LIN {X 0,Y 322.641,Z 978.52,A -85,B 0,C 180,E1 11313.588,E2 11313.588} C_VEL
LIN {X 0,Y 314.07,Z 998.583,A -85,B 0,C 180,E1 11311.867,E2 11311.867} C_VEL
LIN {X 0,Y 304.732,Z 1017.6,A -85,B 0,C 180,E1 11309.836,E2 11309.836} C_VEL
LIN {X 0,Y 294.954,Z 1035.741,A -85,B 0,C 180,E1 11307.468,E2 11307.468} C_VEL
LIN {X 0,Y 285.433,Z 1051.736,A -85,B 0,C 180,E1 11304.898,E2 11304.898} C_VEL
LIN {X 0,Y 275.123,Z 1067.9,A -85,B 0,C 180,E1 11301.721,E2 11301.721} C_VEL
LIN {X 0,Y 265.925,Z 1081.436,A -85,B 0,C 180,E1 11298.438,E2 11298.438} C_VEL
LIN {X 0,Y 256.201,Z 1095.185,A -85,B 0,C 180,E1 11294.314,E2 11294.314} C_VEL
LIN {X 0,Y 248.125,Z 1106.369,A -85,B 0,C 180,E1 11290.148,E2 11290.148} C_VEL
LIN {X 0,Y 240.588,Z 1116.784,A -85,B 0,C 180,E1 11285.288,E2 11285.288} C_VEL
LIN {X 0,Y 234.378,Z 1125.809,A -85,B 0,C 180,E1 11280.002,E2 11280.002} C_VEL
LIN {X 0,Y 229.706,Z 1133.063,A -85,B 0,C 180,E1 11274.427,E2 11274.427} C_VEL
LIN {X 0,Y 226.641,Z 1138.738,A -85,B 0,C 180,E1 11268.788,E2 11268.788} C_VEL
LIN {X 0,Y 224.919,Z 1142.727,A -85,B 0,C 180,E1 11263.105,E2 11263.105} C_VEL
LIN {X 0,Y 224.189,Z 1145.377,A -85,B 0,C 180,E1 11257.432,E2 11257.432} C_VEL
LIN {X 0,Y 224.031,Z 1146.421,A -85,B 0,C 180,E1 11252.303,E2 11252.303} C_VEL
LIN {X 0,Y 224.031,Z 1146.452,A -85,B 0,C 180,E1 11247.954,E2 11247.954} C_VEL
LIN {X 0,Y 224.161,Z 1145.534,A -85,B 0,C 180,E1 11243.083,E2 11243.083} C_VEL
LIN {X 0,Y 224.802,Z 1143.101,A -85,B 0,C 180,E1 11237.413,E2 11237.413} C_VEL
LIN {X 0,Y 226.193,Z 1139.618,A -85,B 0,C 180,E1 11232.242,E2 11232.242} C_VEL
LIN {X 0,Y 229.316,Z 1133.777,A -85,B 0,C 180,E1 11226.078,E2 11226.078} C_VEL
LIN {X 0,Y 233.531,Z 1127.081,A -85,B 0,C 180,E1 11220.785,E2 11220.785} C_VEL
LIN {X 0,Y 239.772,Z 1117.979,A -85,B 0,C 180,E1 11215.236,E2 11215.236} C_VEL
LIN {X 0,Y 247.238,Z 1107.713,A -85,B 0,C 180,E1 11210.285,E2 11210.285} C_VEL
LIN {X 0,Y 255.624,Z 1096.058,A -85,B 0,C 180,E1 11205.875,E2 11205.875} C_VEL
LIN {X 0,Y 265.28,Z 1082.497,A -85,B 0,C 180,E1 11201.731,E2 11201.731} C_VEL
LIN {X 0,Y 274.982,Z 1068.229,A -85,B 0,C 180,E1 11198.243,E2 11198.243} C_VEL
LIN {X 0,Y 285.562,Z 1051.675,A -85,B 0,C 180,E1 11194.983,E2 11194.983} C_VEL
LIN {X 0,Y 294.996,Z 1035.841,A -85,B 0,C 180,E1 11192.44,E2 11192.44} C_VEL
LIN {X 0,Y 304.922,Z 1017.448,A -85,B 0,C 180,E1 11190.041,E2 11190.041} C_VEL
LIN {X 0,Y 313.925,Z 999.165,A -85,B 0,C 180,E1 11188.085,E2 11188.085} C_VEL
LIN {X 0,Y 322.495,Z 979.181,A -85,B 0,C 180,E1 11186.362,E2 11186.362} C_VEL
LIN {X 0,Y 330.224,Z 958.766,A -85,B 0,C 180,E1 11184.929,E2 11184.929} C_VEL
LIN {X 0,Y 336.593,Z 938.741,A -85,B 0,C 180,E1 11183.805,E2 11183.805} C_VEL
LIN {X 0,Y 338.848,Z 930.878,A -85,B 0,C 180,E1 11183.416,E2 11183.416} C_VEL
LIN {X 0,Y 340.313,Z 923.759,A -85,B 0,C 180,E1 11182.949,E2 11182.949} C_VEL
LIN {X 0,Y 342.235,Z 906.193,A -85,B 0,C 180,E1 11181.337,E2 11181.337} C_VEL
LIN {X 0,Y 343.315,Z 898.896,A -85,B 0,C 180,E1 11180.949,E2 11180.949} C_VEL
LIN {X 0,Y 347.119,Z 876.033,A -85,B 0,C 180,E1 11180.35,E2 11180.35} C_VEL
LIN {X 0,Y 351.591,Z 829.528,A -85,B 0,C 180,E1 11179.437,E2 11179.437} C_VEL
LIN {X 0,Y 362.38,Z 710.369,A -85,B 0,C 180,E1 11177.172,E2 11177.172} C_VEL
LIN {X 0,Y 358.599,Z 703.638,A -85,B 0,C 180,E1 11174.534,E2 11174.534} C_VEL
LIN {X 0,Y 355.948,Z 699.091,A -85,B 0,C 180,E1 11172.327,E2 11172.327} C_VEL
LIN {X 0,Y 354.328,Z 696.281,A -85,B 0,C 180,E1 11170.734,E2 11170.734} C_VEL
LIN {X 0,Y 352.108,Z 692.354,A -85,B 0,C 180,E1 11167.999,E2 11167.999} C_VEL
LIN {X 0,Y 350.023,Z 688.483,A -85,B 0,C 180,E1 11163.767,E2 11163.767} C_VEL
LIN {X 0,Y 349.776,Z 687.555,A -85,B 0,C 180,E1 11162.622,E2 11162.622} C_VEL
LIN {X 0,Y 349.89,Z 687.727,A -85,B 0,C 180,E1 11157.38,E2 11157.38} C_VEL
LIN {X 0,Y 351.646,Z 691.826,A -85,B 0,C 180,E1 11153.142,E2 11153.142} C_VEL
LIN {X 0,Y 352.509,Z 693.002,A -85,B 0,C 180,E1 11151.929,E2 11151.929} C_VEL
LIN {X 0,Y 355.354,Z 697.958,A -85,B 0,C 180,E1 11148.723,E2 11148.723} C_VEL
LIN {X 0,Y 357.98,Z 702.565,A -85,B 0,C 180,E1 11146.431,E2 11146.431} C_VEL
LIN {X 0,Y 361.715,Z 709.096,A -85,B 0,C 180,E1 11143.748,E2 11143.748} C_VEL
LIN {X 0,Y 362.516,Z 710.882,A -85,B 0,C 180,E1 11143.207,E2 11143.207} C_VEL
LIN {X 0,Y 346.978,Z 881.346,A -85,B 0,C 180,E1 11139.937,E2 11139.937} C_VEL
LIN {X 0,Y 343.192,Z 905.388,A -85,B 0,C 180,E1 11139.359,E2 11139.359} C_VEL
LIN {X 0,Y 338.384,Z 927.394,A -85,B 0,C 180,E1 11138.689,E2 11138.689} C_VEL
LIN {X 0,Y 332.183,Z 949.393,A -85,B 0,C 180,E1 11137.784,E2 11137.784} C_VEL
LIN {X 0,Y 325.051,Z 970.759,A -85,B 0,C 180,E1 11136.663,E2 11136.663} C_VEL
LIN {X 0,Y 316.962,Z 991.126,A -85,B 0,C 180,E1 11135.298,E2 11135.298} C_VEL
LIN {X 0,Y 307.991,Z 1011.145,A -85,B 0,C 180,E1 11133.638,E2 11133.638} C_VEL
LIN {X 0,Y 298.944,Z 1028.985,A -85,B 0,C 180,E1 11131.801,E2 11131.801} C_VEL
LIN {X 0,Y 288.556,Z 1047.701,A -85,B 0,C 180,E1 11129.436,E2 11129.436} C_VEL
LIN {X 0,Y 278.69,Z 1063.904,A -85,B 0,C 180,E1 11126.901,E2 11126.901} C_VEL
LIN {X 0,Y 267.235,Z 1081.449,A -85,B 0,C 180,E1 11123.495,E2 11123.495} C_VEL
LIN {X 0,Y 257.236,Z 1095.991,A -85,B 0,C 180,E1 11119.971,E2 11119.971} C_VEL
LIN {X 0,Y 247.673,Z 1109.311,A -85,B 0,C 180,E1 11115.938,E2 11115.938} C_VEL
LIN {X 0,Y 238.923,Z 1121.487,A -85,B 0,C 180,E1 11111.392,E2 11111.392} C_VEL
LIN {X 0,Y 231.282,Z 1132.166,A -85,B 0,C 180,E1 11106.318,E2 11106.318} C_VEL
LIN {X 0,Y 225.037,Z 1141.571,A -85,B 0,C 180,E1 11100.727,E2 11100.727} C_VEL
LIN {X 0,Y 220.732,Z 1148.776,A -85,B 0,C 180,E1 11095.201,E2 11095.201} C_VEL
LIN {X 0,Y 217.753,Z 1155.039,A -85,B 0,C 180,E1 11088.937,E2 11088.937} C_VEL
LIN {X 0,Y 216.465,Z 1158.872,A -85,B 0,C 180,E1 11083.625,E2 11083.625} C_VEL
LIN {X 0,Y 216.018,Z 1161.676,A -85,B 0,C 180,E1 11077.981,E2 11077.981} C_VEL
LIN {X 0,Y 215.999,Z 1162.865,A -85,B 0,C 180,E1 11072.918,E2 11072.918} C_VEL
LIN {X 0,Y 216.024,Z 1162.985,A -85,B 0,C 180,E1 11068.408,E2 11068.408} C_VEL
LIN {X 0,Y 215.992,Z 1162.187,A -85,B 0,C 180,E1 11063.887,E2 11063.887} C_VEL
LIN {X 0,Y 216.182,Z 1160.236,A -85,B 0,C 180,E1 11058.798,E2 11058.798} C_VEL
LIN {X 0,Y 217.195,Z 1156.46,A -85,B 0,C 180,E1 11052.864,E2 11052.864} C_VEL
LIN {X 0,Y 219.244,Z 1151.663,A -85,B 0,C 180,E1 11047.475,E2 11047.475} C_VEL
LIN {X 0,Y 223.426,Z 1144.088,A -85,B 0,C 180,E1 11041.097,E2 11041.097} C_VEL
LIN {X 0,Y 228.813,Z 1135.783,A -85,B 0,C 180,E1 11035.677,E2 11035.677} C_VEL
LIN {X 0,Y 235.831,Z 1125.661,A -85,B 0,C 180,E1 11030.499,E2 11030.499} C_VEL
LIN {X 0,Y 244.448,Z 1113.779,A -85,B 0,C 180,E1 11025.617,E2 11025.617} C_VEL
LIN {X 0,Y 253.566,Z 1101.009,A -85,B 0,C 180,E1 11021.477,E2 11021.477} C_VEL
LIN {X 0,Y 264.049,Z 1086.072,A -85,B 0,C 180,E1 11017.563,E2 11017.563} C_VEL
LIN {X 0,Y 274.268,Z 1070.691,A -85,B 0,C 180,E1 11014.337,E2 11014.337} C_VEL
LIN {X 0,Y 285.516,Z 1052.606,A -85,B 0,C 180,E1 11011.297,E2 11011.297} C_VEL
LIN {X 0,Y 295.762,Z 1034.797,A -85,B 0,C 180,E1 11008.885,E2 11008.885} C_VEL
LIN {X 0,Y 305.361,Z 1016.197,A -85,B 0,C 180,E1 11006.862,E2 11006.862} C_VEL
LIN {X 0,Y 314.681,Z 996.301,A -85,B 0,C 180,E1 11005.101,E2 11005.101} C_VEL
LIN {X 0,Y 322.691,Z 976.529,A -85,B 0,C 180,E1 11003.706,E2 11003.706} C_VEL
LIN {X 0,Y 330.129,Z 955.63,A -85,B 0,C 180,E1 11002.518,E2 11002.518} C_VEL
LIN {X 0,Y 336.503,Z 933.853,A -85,B 0,C 180,E1 11001.56,E2 11001.56} C_VEL
LIN {X 0,Y 342.168,Z 909.916,A -85,B 0,C 180,E1 11000.772,E2 11000.772} C_VEL
LIN {X 0,Y 345.989,Z 887.793,A -85,B 0,C 180,E1 11000.215,E2 11000.215} C_VEL
LIN {X 0,Y 349.355,Z 855.488,A -85,B 0,C 180,E1 10999.559,E2 10999.559} C_VEL
LIN {X 0,Y 362.386,Z 710.556,A -85,B 0,C 180,E1 10996.794,E2 10996.794} C_VEL
LIN {X 0,Y 358.527,Z 703.667,A -85,B 0,C 180,E1 10994.123,E2 10994.123} C_VEL
LIN {X 0,Y 355.946,Z 699.194,A -85,B 0,C 180,E1 10991.997,E2 10991.997} C_VEL
LIN {X 0,Y 354.219,Z 696.23,A -85,B 0,C 180,E1 10990.325,E2 10990.325} C_VEL
LIN {X 0,Y 351.914,Z 692.157,A -85,B 0,C 180,E1 10987.509,E2 10987.509} C_VEL
LIN {X 0,Y 349.825,Z 688.191,A -85,B 0,C 180,E1 10983.277,E2 10983.277} C_VEL
LIN {X 0,Y 349.635,Z 687.498,A -85,B 0,C 180,E1 10982.458,E2 10982.458} C_VEL
LIN {X 0,Y 349.707,Z 687.534,A -85,B 0,C 180,E1 10976.722,E2 10976.722} C_VEL
LIN {X 0,Y 351.624,Z 691.848,A -85,B 0,C 180,E1 10972.319,E2 10972.319} C_VEL
LIN {X 0,Y 352.383,Z 692.97,A -85,B 0,C 180,E1 10971.268,E2 10971.268} C_VEL
LIN {X 0,Y 355.185,Z 697.839,A -85,B 0,C 180,E1 10968.141,E2 10968.141} C_VEL
LIN {X 0,Y 358.026,Z 702.794,A -85,B 0,C 180,E1 10965.691,E2 10965.691} C_VEL
LIN {X 0,Y 361.577,Z 708.997,A -85,B 0,C 180,E1 10963.162,E2 10963.162} C_VEL
LIN {X 0,Y 362.209,Z 710.524,A -85,B 0,C 180,E1 10962.727,E2 10962.727} C_VEL
LIN {X 0,Y 347.387,Z 872.495,A -85,B 0,C 180,E1 10959.625,E2 10959.625} C_VEL
LIN {X 0,Y 343.674,Z 896.265,A -85,B 0,C 180,E1 10959.028,E2 10959.028} C_VEL
LIN {X 0,Y 339.285,Z 917.025,A -85,B 0,C 180,E1 10958.329,E2 10958.329} C_VEL
LIN {X 0,Y 333.565,Z 938.122,A -85,B 0,C 180,E1 10957.404,E2 10957.404} C_VEL
LIN {X 0,Y 327.043,Z 958.257,A -85,B 0,C 180,E1 10956.3,E2 10956.3} C_VEL
LIN {X 0,Y 319.125,Z 978.83,A -85,B 0,C 180,E1 10954.889,E2 10954.889} C_VEL
LIN {X 0,Y 310.314,Z 998.919,A -85,B 0,C 180,E1 10953.186,E2 10953.186} C_VEL
LIN {X 0,Y 300.708,Z 1017.933,A -85,B 0,C 180,E1 10951.175,E2 10951.175} C_VEL
LIN {X 0,Y 290.501,Z 1036.276,A -85,B 0,C 180,E1 10948.794,E2 10948.794} C_VEL
LIN {X 0,Y 280.712,Z 1052.181,A -85,B 0,C 180,E1 10946.244,E2 10946.244} C_VEL
LIN {X 0,Y 269.516,Z 1069.043,A -85,B 0,C 180,E1 10942.904,E2 10942.904} C_VEL
LIN {X 0,Y 259.99,Z 1082.505,A -85,B 0,C 180,E1 10939.594,E2 10939.594} C_VEL
LIN {X 0,Y 249.872,Z 1096.119,A -85,B 0,C 180,E1 10935.421,E2 10935.421} C_VEL
LIN {X 0,Y 241.038,Z 1107.802,A -85,B 0,C 180,E1 10930.951,E2 10930.951} C_VEL
LIN {X 0,Y 233.203,Z 1117.989,A -85,B 0,C 180,E1 10925.973,E2 10925.973} C_VEL
LIN {X 0,Y 226.684,Z 1126.902,A -85,B 0,C 180,E1 10920.481,E2 10920.481} C_VEL
LIN {X 0,Y 222.054,Z 1133.666,A -85,B 0,C 180,E1 10915.041,E2 10915.041} C_VEL
LIN {X 0,Y 218.62,Z 1139.557,A -85,B 0,C 180,E1 10908.787,E2 10908.787} C_VEL
LIN {X 0,Y 216.968,Z 1143.185,A -85,B 0,C 180,E1 10903.322,E2 10903.322} C_VEL
LIN {X 0,Y 216.196,Z 1145.743,A -85,B 0,C 180,E1 10897.441,E2 10897.441} C_VEL
LIN {X 0,Y 216.036,Z 1146.721,A -85,B 0,C 180,E1 10892.388,E2 10892.388} C_VEL
LIN {X 0,Y 216.037,Z 1146.751,A -85,B 0,C 180,E1 10887.879,E2 10887.879} C_VEL
LIN {X 0,Y 216.181,Z 1145.835,A -85,B 0,C 180,E1 10882.827,E2 10882.827} C_VEL
LIN {X 0,Y 216.896,Z 1143.405,A -85,B 0,C 180,E1 10876.946,E2 10876.946} C_VEL
LIN {X 0,Y 218.434,Z 1139.923,A -85,B 0,C 180,E1 10871.589,E2 10871.589} C_VEL
LIN {X 0,Y 221.823,Z 1134.084,A -85,B 0,C 180,E1 10865.217,E2 10865.217} C_VEL
LIN {X 0,Y 226.357,Z 1127.39,A -85,B 0,C 180,E1 10859.765,E2 10859.765} C_VEL
LIN {X 0,Y 232.773,Z 1118.619,A -85,B 0,C 180,E1 10854.256,E2 10854.256} C_VEL
LIN {X 0,Y 240.518,Z 1108.538,A -85,B 0,C 180,E1 10849.257,E2 10849.257} C_VEL
LIN {X 0,Y 249.279,Z 1096.988,A -85,B 0,C 180,E1 10844.77,E2 10844.77} C_VEL
LIN {X 0,Y 258.882,Z 1084.199,A -85,B 0,C 180,E1 10840.747,E2 10840.747} C_VEL
LIN {X 0,Y 268.793,Z 1070.2,A -85,B 0,C 180,E1 10837.247,E2 10837.247} C_VEL
LIN {X 0,Y 279.684,Z 1053.979,A -85,B 0,C 180,E1 10833.964,E2 10833.964} C_VEL
LIN {X 0,Y 289.359,Z 1038.337,A -85,B 0,C 180,E1 10831.407,E2 10831.407} C_VEL
LIN {X 0,Y 300.231,Z 1019.071,A -85,B 0,C 180,E1 10828.852,E2 10828.852} C_VEL
LIN {X 0,Y 309.46,Z 1000.923,A -85,B 0,C 180,E1 10826.906,E2 10826.906} C_VEL
LIN {X 0,Y 318.245,Z 981.265,A -85,B 0,C 180,E1 10825.199,E2 10825.199} C_VEL
LIN {X 0,Y 326.15,Z 961.202,A -85,B 0,C 180,E1 10823.781,E2 10823.781} C_VEL
LIN {X 0,Y 333.104,Z 940.106,A -85,B 0,C 180,E1 10822.595,E2 10822.595} C_VEL
LIN {X 0,Y 338.885,Z 919.349,A -85,B 0,C 180,E1 10821.661,E2 10821.661} C_VEL
LIN {X 0,Y 343.315,Z 898.896,A -85,B 0,C 180,E1 10820.949,E2 10820.949} C_VEL
LIN {X 0,Y 344.414,Z 891.512,A -85,B 0,C 180,E1 10820.586,E2 10820.586} C_VEL
LIN {X 0,Y 345.136,Z 873.215,A -85,B 0,C 180,E1 10819.198,E2 10819.198} C_VEL
LIN {X 0,Y 345.634,Z 865.717,A -85,B 0,C 180,E1 10818.884,E2 10818.884} C_VEL
LIN {X 0,Y 359.616,Z 715.682,A -85,B 0,C 180,E1 10816.046,E2 10816.046} C_VEL
LIN {X 0,Y 355.587,Z 708.364,A -85,B 0,C 180,E1 10812.918,E2 10812.918} C_VEL
LIN {X 0,Y 353.04,Z 703.978,A -85,B 0,C 180,E1 10810.443,E2 10810.443} C_VEL
LIN {X 0,Y 350.899,Z 700.114,A -85,B 0,C 180,E1 10807.697,E2 10807.697} C_VEL
LIN {X 0,Y 348.93,Z 696.006,A -85,B 0,C 180,E1 10803.286,E2 10803.286} C_VEL
LIN {X 0,Y 348.728,Z 695.469,A -85,B 0,C 180,E1 10802.301,E2 10802.301} C_VEL
LIN {X 0,Y 348.873,Z 695.622,A -85,B 0,C 180,E1 10797.537,E2 10797.537} C_VEL
LIN {X 0,Y 350.564,Z 699.704,A -85,B 0,C 180,E1 10793.285,E2 10793.285} C_VEL
LIN {X 0,Y 351.343,Z 700.827,A -85,B 0,C 180,E1 10792.149,E2 10792.149} C_VEL
LIN {X 0,Y 354.032,Z 705.658,A -85,B 0,C 180,E1 10789.011,E2 10789.011} C_VEL
LIN {X 0,Y 356.585,Z 710.289,A -85,B 0,C 180,E1 10786.708,E2 10786.708} C_VEL
LIN {X 0,Y 359.758,Z 715.953,A -85,B 0,C 180,E1 10784.338,E2 10784.338} C_VEL
LIN {X 0,Y 344.306,Z 881.021,A -85,B 0,C 180,E1 10781.196,E2 10781.196} C_VEL
LIN {X 0,Y 340.453,Z 905.025,A -85,B 0,C 180,E1 10780.628,E2 10780.628} C_VEL
LIN {X 0,Y 335.385,Z 927.734,A -85,B 0,C 180,E1 10779.95,E2 10779.95} C_VEL
LIN {X 0,Y 329.277,Z 948.882,A -85,B 0,C 180,E1 10779.098,E2 10779.098} C_VEL
LIN {X 0,Y 322.317,Z 969.404,A -85,B 0,C 180,E1 10778.052,E2 10778.052} C_VEL
LIN {X 0,Y 314.028,Z 989.917,A -85,B 0,C 180,E1 10776.719,E2 10776.719} C_VEL
LIN {X 0,Y 304.817,Z 1010.101,A -85,B 0,C 180,E1 10775.09,E2 10775.09} C_VEL
LIN {X 0,Y 295.23,Z 1028.514,A -85,B 0,C 180,E1 10773.229,E2 10773.229} C_VEL
LIN {X 0,Y 284.787,Z 1046.833,A -85,B 0,C 180,E1 10770.952,E2 10770.952} C_VEL
LIN {X 0,Y 274.573,Z 1063.082,A -85,B 0,C 180,E1 10768.442,E2 10768.442} C_VEL
LIN {X 0,Y 263.074,Z 1080.141,A -85,B 0,C 180,E1 10765.179,E2 10765.179} C_VEL
LIN {X 0,Y 253.046,Z 1094.112,A -85,B 0,C 180,E1 10761.841,E2 10761.841} C_VEL
LIN {X 0,Y 242.409,Z 1108.35,A -85,B 0,C 180,E1 10757.588,E2 10757.588} C_VEL
LIN {X 0,Y 233.113,Z 1120.589,A -85,B 0,C 180,E1 10752.998,E2 10752.998} C_VEL
LIN {X 0,Y 224.926,Z 1131.382,A -85,B 0,C 180,E1 10747.839,E2 10747.839} C_VEL
LIN {X 0,Y 218.161,Z 1140.894,A -85,B 0,C 180,E1 10742.116,E2 10742.116} C_VEL
LIN {X 0,Y 213.43,Z 1148.152,A -85,B 0,C 180,E1 10736.426,E2 10736.426} C_VEL
LIN {X 0,Y 210.207,Z 1154.229,A -85,B 0,C 180,E1 10730.317,E2 10730.317} C_VEL
LIN {X 0,Y 208.585,Z 1158.399,A -85,B 0,C 180,E1 10724.433,E2 10724.433} C_VEL
LIN {X 0,Y 208.057,Z 1161.14,A -85,B 0,C 180,E1 10718.846,E2 10718.846} C_VEL
LIN {X 0,Y 208.001,Z 1162.54,A -85,B 0,C 180,E1 10713.306,E2 10713.306} C_VEL
LIN {X 0,Y 208.029,Z 1162.707,A -85,B 0,C 180,E1 10708.608,E2 10708.608} C_VEL
LIN {X 0,Y 207.995,Z 1161.957,A -85,B 0,C 180,E1 10703.929,E2 10703.929} C_VEL
LIN {X 0,Y 208.144,Z 1160.292,A -85,B 0,C 180,E1 10699.201,E2 10699.201} C_VEL
LIN {X 0,Y 209.055,Z 1157.012,A -85,B 0,C 180,E1 10693.323,E2 10693.323} C_VEL
LIN {X 0,Y 211.328,Z 1151.881,A -85,B 0,C 180,E1 10687.171,E2 10687.171} C_VEL
LIN {X 0,Y 215.256,Z 1145.232,A -85,B 0,C 180,E1 10681.113,E2 10681.113} C_VEL
LIN {X 0,Y 220.698,Z 1137.149,A -85,B 0,C 180,E1 10675.506,E2 10675.506} C_VEL
LIN {X 0,Y 228.236,Z 1126.942,A -85,B 0,C 180,E1 10669.91,E2 10669.91} C_VEL
LIN {X 0,Y 236.315,Z 1116.281,A -85,B 0,C 180,E1 10665.3,E2 10665.3} C_VEL
LIN {X 0,Y 246.503,Z 1102.835,A -85,B 0,C 180,E1 10660.666,E2 10660.666} C_VEL
LIN {X 0,Y 256.84,Z 1088.844,A -85,B 0,C 180,E1 10656.834,E2 10656.834} C_VEL
LIN {X 0,Y 267.816,Z 1073.089,A -85,B 0,C 180,E1 10653.4,E2 10653.4} C_VEL
LIN {X 0,Y 278.917,Z 1056.225,A -85,B 0,C 180,E1 10650.441,E2 10650.441} C_VEL
LIN {X 0,Y 289.106,Z 1039.202,A -85,B 0,C 180,E1 10648.056,E2 10648.056} C_VEL
LIN {X 0,Y 299.546,Z 1020.253,A -85,B 0,C 180,E1 10645.897,E2 10645.897} C_VEL
LIN {X 0,Y 308.98,Z 1000.939,A -85,B 0,C 180,E1 10644.138,E2 10644.138} C_VEL
LIN {X 0,Y 318.643,Z 978.426,A -85,B 0,C 180,E1 10642.508,E2 10642.508} C_VEL
LIN {X 0,Y 326.708,Z 956.546,A -85,B 0,C 180,E1 10641.266,E2 10641.266} C_VEL
LIN {X 0,Y 333.415,Z 934.284,A -85,B 0,C 180,E1 10640.298,E2 10640.298} C_VEL
LIN {X 0,Y 339.086,Z 911.171,A -85,B 0,C 180,E1 10639.543,E2 10639.543} C_VEL
LIN {X 0,Y 343.088,Z 888.779,A -85,B 0,C 180,E1 10638.984,E2 10638.984} C_VEL
LIN {X 0,Y 346.52,Z 857.614,A -85,B 0,C 180,E1 10638.352,E2 10638.352} C_VEL
LIN {X 0,Y 359.576,Z 715.777,A -85,B 0,C 180,E1 10635.647,E2 10635.647} C_VEL
LIN {X 0,Y 355.316,Z 708.035,A -85,B 0,C 180,E1 10632.348,E2 10632.348} C_VEL
LIN {X 0,Y 352.926,Z 703.924,A -85,B 0,C 180,E1 10630.034,E2 10630.034} C_VEL
LIN {X 0,Y 350.821,Z 700.035,A -85,B 0,C 180,E1 10627.368,E2 10627.368} C_VEL
LIN {X 0,Y 348.762,Z 695.893,A -85,B 0,C 180,E1 10622.958,E2 10622.958} C_VEL
LIN {X 0,Y 348.575,Z 695.405,A -85,B 0,C 180,E1 10622.137,E2 10622.137} C_VEL
LIN {X 0,Y 348.719,Z 695.594,A -85,B 0,C 180,E1 10616.712,E2 10616.712} C_VEL
LIN {X 0,Y 350.538,Z 699.727,A -85,B 0,C 180,E1 10612.46,E2 10612.46} C_VEL
LIN {X 0,Y 351.271,Z 700.935,A -85,B 0,C 180,E1 10611.405,E2 10611.405} C_VEL
LIN {X 0,Y 353.862,Z 705.543,A -85,B 0,C 180,E1 10608.427,E2 10608.427} C_VEL
LIN {X 0,Y 356.725,Z 710.693,A -85,B 0,C 180,E1 10605.886,E2 10605.886} C_VEL
LIN {X 0,Y 359.468,Z 715.577,A -85,B 0,C 180,E1 10603.855,E2 10603.855} C_VEL
LIN {X 0,Y 344.671,Z 872.923,A -85,B 0,C 180,E1 10600.87,E2 10600.87} C_VEL
LIN {X 0,Y 340.891,Z 896.579,A -85,B 0,C 180,E1 10600.285,E2 10600.285} C_VEL
LIN {X 0,Y 336.406,Z 917.337,A -85,B 0,C 180,E1 10599.598,E2 10599.598} C_VEL
LIN {X 0,Y 330.559,Z 938.431,A -85,B 0,C 180,E1 10598.691,E2 10598.691} C_VEL
LIN {X 0,Y 323.888,Z 958.566,A -85,B 0,C 180,E1 10597.606,E2 10597.606} C_VEL
LIN {X 0,Y 315.779,Z 979.139,A -85,B 0,C 180,E1 10596.217,E2 10596.217} C_VEL
LIN {X 0,Y 306.752,Z 999.202,A -85,B 0,C 180,E1 10594.541,E2 10594.541} C_VEL
LIN {X 0,Y 296.844,Z 1018.287,A -85,B 0,C 180,E1 10592.547,E2 10592.547} C_VEL
LIN {X 0,Y 286.349,Z 1036.586,A -85,B 0,C 180,E1 10590.194,E2 10590.194} C_VEL
LIN {X 0,Y 276.292,Z 1052.408,A -85,B 0,C 180,E1 10587.674,E2 10587.674} C_VEL
LIN {X 0,Y 264.638,Z 1069.354,A -85,B 0,C 180,E1 10584.324,E2 10584.324} C_VEL
LIN {X 0,Y 254.723,Z 1082.817,A -85,B 0,C 180,E1 10581.007,E2 10581.007} C_VEL
LIN {X 0,Y 244.136,Z 1096.432,A -85,B 0,C 180,E1 10576.804,E2 10576.804} C_VEL
LIN {X 0,Y 234.851,Z 1108.115,A -85,B 0,C 180,E1 10572.275,E2 10572.275} C_VEL
LIN {X 0,Y 226.558,Z 1118.301,A -85,B 0,C 180,E1 10567.202,E2 10567.202} C_VEL
LIN {X 0,Y 219.6,Z 1127.213,A -85,B 0,C 180,E1 10561.575,E2 10561.575} C_VEL
LIN {X 0,Y 214.6,Z 1134.007,A -85,B 0,C 180,E1 10555.943,E2 10555.943} C_VEL
LIN {X 0,Y 210.971,Z 1139.749,A -85,B 0,C 180,E1 10549.664,E2 10549.664} C_VEL
LIN {X 0,Y 209.077,Z 1143.49,A -85,B 0,C 180,E1 10543.835,E2 10543.835} C_VEL
LIN {X 0,Y 208.221,Z 1146.045,A -85,B 0,C 180,E1 10537.728,E2 10537.728} C_VEL
LIN {X 0,Y 208.042,Z 1147.021,A -85,B 0,C 180,E1 10532.48,E2 10532.48} C_VEL
LIN {X 0,Y 208.042,Z 1147.051,A -85,B 0,C 180,E1 10527.797,E2 10527.797} C_VEL
LIN {X 0,Y 208.188,Z 1146.2,A -85,B 0,C 180,E1 10522.827,E2 10522.827} C_VEL
LIN {X 0,Y 208.892,Z 1144.015,A -85,B 0,C 180,E1 10517,E2 10517} C_VEL
LIN {X 0,Y 210.584,Z 1140.427,A -85,B 0,C 180,E1 10511.164,E2 10511.164} C_VEL
LIN {X 0,Y 214.001,Z 1134.978,A -85,B 0,C 180,E1 10504.839,E2 10504.839} C_VEL
LIN {X 0,Y 218.724,Z 1128.383,A -85,B 0,C 180,E1 10499.204,E2 10499.204} C_VEL
LIN {X 0,Y 225.757,Z 1119.375,A -85,B 0,C 180,E1 10493.281,E2 10493.281} C_VEL
LIN {X 0,Y 233.453,Z 1109.852,A -85,B 0,C 180,E1 10488.406,E2 10488.406} C_VEL
LIN {X 0,Y 243.031,Z 1097.919,A -85,B 0,C 180,E1 10483.608,E2 10483.608} C_VEL
LIN {X 0,Y 253.166,Z 1085.046,A -85,B 0,C 180,E1 10479.484,E2 10479.484} C_VEL
LIN {X 0,Y 263.895,Z 1070.505,A -85,B 0,C 180,E1 10475.825,E2 10475.825} C_VEL
LIN {X 0,Y 275.183,Z 1054.283,A -85,B 0,C 180,E1 10472.547,E2 10472.547} C_VEL
LIN {X 0,Y 285.182,Z 1038.64,A -85,B 0,C 180,E1 10470.004,E2 10470.004} C_VEL
LIN {X 0,Y 296.384,Z 1019.372,A -85,B 0,C 180,E1 10467.472,E2 10467.472} C_VEL
LIN {X 0,Y 305.871,Z 1001.222,A -85,B 0,C 180,E1 10465.55,E2 10465.55} C_VEL
LIN {X 0,Y 314.884,Z 981.563,A -85,B 0,C 180,E1 10463.867,E2 10463.867} C_VEL
LIN {X 0,Y 322.982,Z 961.498,A -85,B 0,C 180,E1 10462.472,E2 10462.472} C_VEL
LIN {X 0,Y 330.009,Z 940.687,A -85,B 0,C 180,E1 10461.32,E2 10461.32} C_VEL
LIN {X 0,Y 336.006,Z 919.64,A -85,B 0,C 180,E1 10460.389,E2 10460.389} C_VEL
LIN {X 0,Y 340.804,Z 897.8,A -85,B 0,C 180,E1 10459.651,E2 10459.651} C_VEL
LIN {X 0,Y 344.627,Z 874.674,A -85,B 0,C 180,E1 10459.067,E2 10459.067} C_VEL
LIN {X 0,Y 345.634,Z 865.717,A -85,B 0,C 180,E1 10458.884,E2 10458.884} C_VEL
LIN {X 0,Y 346.123,Z 858.188,A -85,B 0,C 180,E1 10458.579,E2 10458.579} C_VEL
LIN {X 0,Y 346.022,Z 838.591,A -85,B 0,C 180,E1 10457.217,E2 10457.217} C_VEL
LIN {X 0,Y 346.402,Z 832.101,A -85,B 0,C 180,E1 10456.978,E2 10456.978} C_VEL
LIN {X 0,Y 356.97,Z 721.273,A -85,B 0,C 180,E1 10454.91,E2 10454.91} C_VEL
LIN {X 0,Y 353.616,Z 715.07,A -85,B 0,C 180,E1 10452.078,E2 10452.078} C_VEL
LIN {X 0,Y 351.761,Z 711.675,A -85,B 0,C 180,E1 10450.151,E2 10450.151} C_VEL
LIN {X 0,Y 349.812,Z 707.993,A -85,B 0,C 180,E1 10447.556,E2 10447.556} C_VEL
LIN {X 0,Y 347.91,Z 703.899,A -85,B 0,C 180,E1 10443.131,E2 10443.131} C_VEL
LIN {X 0,Y 347.721,Z 703.395,A -85,B 0,C 180,E1 10442.143,E2 10442.143} C_VEL
LIN {X 0,Y 347.859,Z 703.517,A -85,B 0,C 180,E1 10437.694,E2 10437.694} C_VEL
LIN {X 0,Y 349.588,Z 707.703,A -85,B 0,C 180,E1 10433.266,E2 10433.266} C_VEL
LIN {X 0,Y 350.289,Z 708.92,A -85,B 0,C 180,E1 10432.208,E2 10432.208} C_VEL
LIN {X 0,Y 352.795,Z 713.514,A -85,B 0,C 180,E1 10429.22,E2 10429.22} C_VEL
LIN {X 0,Y 355.199,Z 718.012,A -85,B 0,C 180,E1 10426.986,E2 10426.986} C_VEL
LIN {X 0,Y 357.097,Z 721.646,A -85,B 0,C 180,E1 10425.466,E2 10425.466} C_VEL
LIN {X 0,Y 341.795,Z 880.76,A -85,B 0,C 180,E1 10422.472,E2 10422.472} C_VEL
LIN {X 0,Y 337.855,Z 904.805,A -85,B 0,C 180,E1 10421.914,E2 10421.914} C_VEL
LIN {X 0,Y 332.831,Z 926.949,A -85,B 0,C 180,E1 10421.27,E2 10421.27} C_VEL
LIN {X 0,Y 326.767,Z 947.687,A -85,B 0,C 180,E1 10420.464,E2 10420.464} C_VEL
LIN {X 0,Y 319.369,Z 969.106,A -85,B 0,C 180,E1 10419.404,E2 10419.404} C_VEL
LIN {X 0,Y 310.836,Z 989.747,A -85,B 0,C 180,E1 10418.091,E2 10418.091} C_VEL
LIN {X 0,Y 301.455,Z 1009.798,A -85,B 0,C 180,E1 10416.504,E2 10416.504} C_VEL
LIN {X 0,Y 291.52,Z 1028.375,A -85,B 0,C 180,E1 10414.656,E2 10414.656} C_VEL
LIN {X 0,Y 280.501,Z 1047.087,A -85,B 0,C 180,E1 10412.348,E2 10412.348} C_VEL
LIN {X 0,Y 269.976,Z 1063.287,A -85,B 0,C 180,E1 10409.856,E2 10409.856} C_VEL
LIN {X 0,Y 257.766,Z 1080.689,A -85,B 0,C 180,E1 10406.508,E2 10406.508} C_VEL
LIN {X 0,Y 247.38,Z 1094.584,A -85,B 0,C 180,E1 10403.156,E2 10403.156} C_VEL
LIN {X 0,Y 236.308,Z 1108.685,A -85,B 0,C 180,E1 10398.863,E2 10398.863} C_VEL
LIN {X 0,Y 226.596,Z 1120.861,A -85,B 0,C 180,E1 10394.2,E2 10394.2} C_VEL
LIN {X 0,Y 217.99,Z 1131.54,A -85,B 0,C 180,E1 10388.93,E2 10388.93} C_VEL
LIN {X 0,Y 210.837,Z 1140.947,A -85,B 0,C 180,E1 10383.049,E2 10383.049} C_VEL
LIN {X 0,Y 205.813,Z 1148.155,A -85,B 0,C 180,E1 10377.171,E2 10377.171} C_VEL
LIN {X 0,Y 202.251,Z 1154.352,A -85,B 0,C 180,E1 10370.548,E2 10370.548} C_VEL
LIN {X 0,Y 200.628,Z 1158.26,A -85,B 0,C 180,E1 10364.724,E2 10364.724} C_VEL
LIN {X 0,Y 200.051,Z 1161.072,A -85,B 0,C 180,E1 10358.623,E2 10358.623} C_VEL
LIN {X 0,Y 200.006,Z 1162.265,A -85,B 0,C 180,E1 10353.152,E2 10353.152} C_VEL
LIN {X 0,Y 200.034,Z 1162.406,A -85,B 0,C 180,E1 10348.536,E2 10348.536} C_VEL
LIN {X 0,Y 200.004,Z 1161.656,A -85,B 0,C 180,E1 10343.685,E2 10343.685} C_VEL
LIN {X 0,Y 200.182,Z 1159.987,A -85,B 0,C 180,E1 10338.767,E2 10338.767} C_VEL
LIN {X 0,Y 201.289,Z 1156.488,A -85,B 0,C 180,E1 10332.361,E2 10332.361} C_VEL
LIN {X 0,Y 203.722,Z 1151.57,A -85,B 0,C 180,E1 10326.268,E2 10326.268} C_VEL
LIN {X 0,Y 208.218,Z 1144.553,A -85,B 0,C 180,E1 10319.72,E2 10319.72} C_VEL
LIN {X 0,Y 214.165,Z 1136.416,A -85,B 0,C 180,E1 10313.966,E2 10313.966} C_VEL
LIN {X 0,Y 222.703,Z 1125.571,A -85,B 0,C 180,E1 10308.012,E2 10308.012} C_VEL
LIN {X 0,Y 231.757,Z 1114.347,A -85,B 0,C 180,E1 10303.187,E2 10303.187} C_VEL
LIN {X 0,Y 242.236,Z 1101.091,A -85,B 0,C 180,E1 10298.727,E2 10298.727} C_VEL
LIN {X 0,Y 253.383,Z 1086.583,A -85,B 0,C 180,E1 10294.836,E2 10294.836} C_VEL
LIN {X 0,Y 264.555,Z 1071.017,A -85,B 0,C 180,E1 10291.548,E2 10291.548} C_VEL
LIN {X 0,Y 276.846,Z 1052.66,A -85,B 0,C 180,E1 10288.472,E2 10288.472} C_VEL
LIN {X 0,Y 286.89,Z 1036.273,A -85,B 0,C 180,E1 10286.27,E2 10286.27} C_VEL
LIN {X 0,Y 297.416,Z 1017.291,A -85,B 0,C 180,E1 10284.213,E2 10284.213} C_VEL
LIN {X 0,Y 306.519,Z 998.992,A -85,B 0,C 180,E1 10282.609,E2 10282.609} C_VEL
LIN {X 0,Y 315.692,Z 977.93,A -85,B 0,C 180,E1 10281.132,E2 10281.132} C_VEL
LIN {X 0,Y 323.442,Z 957.372,A -85,B 0,C 180,E1 10279.987,E2 10279.987} C_VEL
LIN {X 0,Y 330.281,Z 935.458,A -85,B 0,C 180,E1 10279.041,E2 10279.041} C_VEL
LIN {X 0,Y 336.111,Z 912.686,A -85,B 0,C 180,E1 10278.299,E2 10278.299} C_VEL
LIN {X 0,Y 340.4,Z 889.439,A -85,B 0,C 180,E1 10277.726,E2 10277.726} C_VEL
LIN {X 0,Y 343.879,Z 859.33,A -85,B 0,C 180,E1 10277.118,E2 10277.118} C_VEL
LIN {X 0,Y 356.924,Z 721.387,A -85,B 0,C 180,E1 10274.52,E2 10274.52} C_VEL
LIN {X 0,Y 353.434,Z 714.872,A -85,B 0,C 180,E1 10271.587,E2 10271.587} C_VEL
LIN {X 0,Y 351.569,Z 711.51,A -85,B 0,C 180,E1 10269.659,E2 10269.659} C_VEL
LIN {X 0,Y 349.615,Z 707.792,A -85,B 0,C 180,E1 10267.063,E2 10267.063} C_VEL
LIN {X 0,Y 347.71,Z 703.594,A -85,B 0,C 180,E1 10262.637,E2 10262.637} C_VEL
LIN {X 0,Y 347.508,Z 703.319,A -85,B 0,C 180,E1 10257.691,E2 10257.691} C_VEL
LIN {X 0,Y 347.727,Z 703.685,A -85,B 0,C 180,E1 10256.703,E2 10256.703} C_VEL
LIN {X 0,Y 349.676,Z 707.857,A -85,B 0,C 180,E1 10252.276,E2 10252.276} C_VEL
LIN {X 0,Y 352.549,Z 713.247,A -85,B 0,C 180,E1 10248.715,E2 10248.715} C_VEL
LIN {X 0,Y 355.331,Z 718.414,A -85,B 0,C 180,E1 10246.162,E2 10246.162} C_VEL
LIN {X 0,Y 356.801,Z 721.336,A -85,B 0,C 180,E1 10244.987,E2 10244.987} C_VEL
LIN {X 0,Y 342.133,Z 873.245,A -85,B 0,C 180,E1 10242.135,E2 10242.135} C_VEL
LIN {X 0,Y 338.291,Z 896.811,A -85,B 0,C 180,E1 10241.563,E2 10241.563} C_VEL
LIN {X 0,Y 333.72,Z 917.54,A -85,B 0,C 180,E1 10240.893,E2 10240.893} C_VEL
LIN {X 0,Y 327.723,Z 938.741,A -85,B 0,C 180,E1 10240.001,E2 10240.001} C_VEL
LIN {X 0,Y 320.904,Z 958.876,A -85,B 0,C 180,E1 10238.936,E2 10238.936} C_VEL
LIN {X 0,Y 312.607,Z 979.448,A -85,B 0,C 180,E1 10237.573,E2 10237.573} C_VEL
LIN {X 0,Y 303.354,Z 999.511,A -85,B 0,C 180,E1 10235.924,E2 10235.924} C_VEL
LIN {X 0,Y 293.347,Z 1018.299,A -85,B 0,C 180,E1 10233.992,E2 10233.992} C_VEL
LIN {X 0,Y 282.376,Z 1036.896,A -85,B 0,C 180,E1 10231.633,E2 10231.633} C_VEL
LIN {X 0,Y 271.963,Z 1052.765,A -85,B 0,C 180,E1 10229.126,E2 10229.126} C_VEL
LIN {X 0,Y 259.928,Z 1069.666,A -85,B 0,C 180,E1 10225.797,E2 10225.797} C_VEL
LIN {X 0,Y 249.617,Z 1083.128,A -85,B 0,C 180,E1 10222.478,E2 10222.478} C_VEL
LIN {X 0,Y 238.551,Z 1096.744,A -85,B 0,C 180,E1 10218.252,E2 10218.252} C_VEL
LIN {X 0,Y 228.797,Z 1108.427,A -85,B 0,C 180,E1 10213.669,E2 10213.669} C_VEL
LIN {X 0,Y 220.021,Z 1118.613,A -85,B 0,C 180,E1 10208.506,E2 10208.506} C_VEL
LIN {X 0,Y 212.604,Z 1127.524,A -85,B 0,C 180,E1 10202.741,E2 10202.741} C_VEL
LIN {X 0,Y 207.248,Z 1134.286,A -85,B 0,C 180,E1 10196.969,E2 10196.969} C_VEL
LIN {X 0,Y 203.287,Z 1140.056,A -85,B 0,C 180,E1 10190.44,E2 10190.44} C_VEL
LIN {X 0,Y 201.2,Z 1143.795,A -85,B 0,C 180,E1 10184.388,E2 10184.388} C_VEL
LIN {X 0,Y 200.251,Z 1146.347,A -85,B 0,C 180,E1 10178.037,E2 10178.037} C_VEL
LIN {X 0,Y 200.047,Z 1147.321,A -85,B 0,C 180,E1 10172.579,E2 10172.579} C_VEL
LIN {X 0,Y 200.047,Z 1147.373,A -85,B 0,C 180,E1 10167.996,E2 10167.996} C_VEL
LIN {X 0,Y 200.179,Z 1146.63,A -85,B 0,C 180,E1 10163.116,E2 10163.116} C_VEL
LIN {X 0,Y 200.885,Z 1144.62,A -85,B 0,C 180,E1 10157.058,E2 10157.058} C_VEL
LIN {X 0,Y 202.747,Z 1140.931,A -85,B 0,C 180,E1 10150.707,E2 10150.707} C_VEL
LIN {X 0,Y 206.207,Z 1135.845,A -85,B 0,C 180,E1 10144.407,E2 10144.407} C_VEL
LIN {X 0,Y 211.385,Z 1129.034,A -85,B 0,C 180,E1 10138.33,E2 10138.33} C_VEL
LIN {X 0,Y 218.447,Z 1120.578,A -85,B 0,C 180,E1 10132.501,E2 10132.501} C_VEL
LIN {X 0,Y 226.883,Z 1110.663,A -85,B 0,C 180,E1 10127.261,E2 10127.261} C_VEL
LIN {X 0,Y 236.888,Z 1098.849,A -85,B 0,C 180,E1 10122.385,E2 10122.385} C_VEL
LIN {X 0,Y 247.179,Z 1086.333,A -85,B 0,C 180,E1 10118.303,E2 10118.303} C_VEL
LIN {X 0,Y 257.914,Z 1072.475,A -85,B 0,C 180,E1 10114.729,E2 10114.729} C_VEL
LIN {X 0,Y 268.86,Z 1057.515,A -85,B 0,C 180,E1 10111.612,E2 10111.612} C_VEL
LIN {X 0,Y 279.777,Z 1041.136,A -85,B 0,C 180,E1 10108.887,E2 10108.887} C_VEL
LIN {X 0,Y 290.529,Z 1023.634,A -85,B 0,C 180,E1 10106.519,E2 10106.519} C_VEL
LIN {X 0,Y 300.697,Z 1004.903,A -85,B 0,C 180,E1 10104.493,E2 10104.493} C_VEL
LIN {X 0,Y 310.367,Z 984.938,A -85,B 0,C 180,E1 10102.743,E2 10102.743} C_VEL
LIN {X 0,Y 318.395,Z 965.784,A -85,B 0,C 180,E1 10101.393,E2 10101.393} C_VEL
LIN {X 0,Y 326.394,Z 943.451,A -85,B 0,C 180,E1 10100.13,E2 10100.13} C_VEL
LIN {X 0,Y 332.062,Z 924.35,A -85,B 0,C 180,E1 10099.271,E2 10099.271} C_VEL
LIN {X 0,Y 337.697,Z 900.594,A -85,B 0,C 180,E1 10098.444,E2 10098.444} C_VEL
LIN {X 0,Y 341.548,Z 878.704,A -85,B 0,C 180,E1 10097.882,E2 10097.882} C_VEL
LIN {X 0,Y 345.155,Z 845.358,A -85,B 0,C 180,E1 10097.226,E2 10097.226} C_VEL
LIN {X 0,Y 346.402,Z 832.101,A -85,B 0,C 180,E1 10096.978,E2 10096.978} C_VEL
LIN {X 0,Y 346.83,Z 824.559,A -85,B 0,C 180,E1 10096.68,E2 10096.68} C_VEL
LIN {X 0,Y 346.999,Z 804.975,A -85,B 0,C 180,E1 10095.316,E2 10095.316} C_VEL
LIN {X 0,Y 347.441,Z 798.487,A -85,B 0,C 180,E1 10095.08,E2 10095.08} C_VEL
LIN {X 0,Y 354.461,Z 726.877,A -85,B 0,C 180,E1 10093.756,E2 10093.756} C_VEL
LIN {X 0,Y 351.5,Z 721.267,A -85,B 0,C 180,E1 10090.987,E2 10090.987} C_VEL
LIN {X 0,Y 350.149,Z 718.825,A -85,B 0,C 180,E1 10089.451,E2 10089.451} C_VEL
LIN {X 0,Y 348.618,Z 715.752,A -85,B 0,C 180,E1 10087.25,E2 10087.25} C_VEL
LIN {X 0,Y 346.87,Z 711.606,A -85,B 0,C 180,E1 10082.809,E2 10082.809} C_VEL
LIN {X 0,Y 346.779,Z 711.336,A -85,B 0,C 180,E1 10078.183,E2 10078.183} C_VEL
LIN {X 0,Y 349.028,Z 716.474,A -85,B 0,C 180,E1 10072.594,E2 10072.594} C_VEL
LIN {X 0,Y 351.489,Z 721.212,A -85,B 0,C 180,E1 10069.511,E2 10069.511} C_VEL
LIN {X 0,Y 353.912,Z 725.906,A -85,B 0,C 180,E1 10067.187,E2 10067.187} C_VEL
LIN {X 0,Y 354.566,Z 727.372,A -85,B 0,C 180,E1 10066.615,E2 10066.615} C_VEL
LIN {X 0,Y 339.443,Z 880.607,A -85,B 0,C 180,E1 10063.765,E2 10063.765} C_VEL
LIN {X 0,Y 335.421,Z 904.63,A -85,B 0,C 180,E1 10063.218,E2 10063.218} C_VEL
LIN {X 0,Y 330.331,Z 926.658,A -85,B 0,C 180,E1 10062.594,E2 10062.594} C_VEL
LIN {X 0,Y 324.151,Z 947.391,A -85,B 0,C 180,E1 10061.812,E2 10061.812} C_VEL
LIN {X 0,Y 316.603,Z 968.808,A -85,B 0,C 180,E1 10060.781,E2 10060.781} C_VEL
LIN {X 0,Y 307.942,Z 989.317,A -85,B 0,C 180,E1 10059.51,E2 10059.51} C_VEL
LIN {X 0,Y 298.297,Z 1009.465,A -85,B 0,C 180,E1 10057.951,E2 10057.951} C_VEL
LIN {X 0,Y 288.171,Z 1027.929,A -85,B 0,C 180,E1 10056.152,E2 10056.152} C_VEL
LIN {X 0,Y 276.6,Z 1047.021,A -85,B 0,C 180,E1 10053.832,E2 10053.832} C_VEL
LIN {X 0,Y 265.548,Z 1063.492,A -85,B 0,C 180,E1 10051.319,E2 10051.319} C_VEL
LIN {X 0,Y 253.13,Z 1080.553,A -85,B 0,C 180,E1 10048.043,E2 10048.043} C_VEL
LIN {X 0,Y 241.849,Z 1095.057,A -85,B 0,C 180,E1 10044.532,E2 10044.532} C_VEL
LIN {X 0,Y 230.873,Z 1108.372,A -85,B 0,C 180,E1 10040.432,E2 10040.432} C_VEL
LIN {X 0,Y 220.661,Z 1120.548,A -85,B 0,C 180,E1 10035.719,E2 10035.719} C_VEL
LIN {X 0,Y 211.529,Z 1131.227,A -85,B 0,C 180,E1 10030.358,E2 10030.358} C_VEL
LIN {X 0,Y 203.873,Z 1140.634,A -85,B 0,C 180,E1 10024.332,E2 10024.332} C_VEL
LIN {X 0,Y 198.441,Z 1147.844,A -85,B 0,C 180,E1 10018.269,E2 10018.269} C_VEL
LIN {X 0,Y 194.418,Z 1154.259,A -85,B 0,C 180,E1 10011.1,E2 10011.1} C_VEL
LIN {X 0,Y 192.701,Z 1158.039,A -85,B 0,C 180,E1 10005.187,E2 10005.187} C_VEL
LIN {X 0,Y 192.055,Z 1160.851,A -85,B 0,C 180,E1 9998.683,E2 9998.683} C_VEL
LIN {X 0,Y 192.013,Z 1161.989,A -85,B 0,C 180,E1 9992.984,E2 9992.984} C_VEL
LIN {X 0,Y 192.038,Z 1162.085,A -85,B 0,C 180,E1 9988.209,E2 9988.209} C_VEL
LIN {X 0,Y 192.008,Z 1161.354,A -85,B 0,C 180,E1 9983.421,E2 9983.421} C_VEL
LIN {X 0,Y 192.226,Z 1159.682,A -85,B 0,C 180,E1 9978.295,E2 9978.295} C_VEL
LIN {X 0,Y 193.476,Z 1156.179,A -85,B 0,C 180,E1 9971.624,E2 9971.624} C_VEL
LIN {X 0,Y 196.15,Z 1151.258,A -85,B 0,C 180,E1 9965.291,E2 9965.291} C_VEL
LIN {X 0,Y 200.79,Z 1144.604,A -85,B 0,C 180,E1 9958.809,E2 9958.809} C_VEL
LIN {X 0,Y 207.267,Z 1136.315,A -85,B 0,C 180,E1 9952.745,E2 9952.745} C_VEL
LIN {X 0,Y 216.096,Z 1125.781,A -85,B 0,C 180,E1 9946.78,E2 9946.78} C_VEL
LIN {X 0,Y 225.581,Z 1114.617,A -85,B 0,C 180,E1 9941.871,E2 9941.871} C_VEL
LIN {X 0,Y 236.504,Z 1101.488,A -85,B 0,C 180,E1 9937.362,E2 9937.362} C_VEL
LIN {X 0,Y 248.068,Z 1087.108,A -85,B 0,C 180,E1 9933.452,E2 9933.452} C_VEL
LIN {X 0,Y 259.967,Z 1071.155,A -85,B 0,C 180,E1 9930.073,E2 9930.073} C_VEL
LIN {X 0,Y 271.984,Z 1053.912,A -85,B 0,C 180,E1 9927.171,E2 9927.171} C_VEL
LIN {X 0,Y 282.357,Z 1037.548,A -85,B 0,C 180,E1 9924.968,E2 9924.968} C_VEL
LIN {X 0,Y 293.923,Z 1017.403,A -85,B 0,C 180,E1 9922.795,E2 9922.795} C_VEL
LIN {X 0,Y 303.068,Z 999.499,A -85,B 0,C 180,E1 9921.249,E2 9921.249} C_VEL
LIN {X 0,Y 312.854,Z 977.618,A -85,B 0,C 180,E1 9919.744,E2 9919.744} C_VEL
LIN {X 0,Y 320.764,Z 957.061,A -85,B 0,C 180,E1 9918.628,E2 9918.628} C_VEL
LIN {X 0,Y 327.814,Z 934.876,A -85,B 0,C 180,E1 9917.697,E2 9917.697} C_VEL
LIN {X 0,Y 333.725,Z 912.11,A -85,B 0,C 180,E1 9916.979,E2 9916.979} C_VEL
LIN {X 0,Y 338.036,Z 889.121,A -85,B 0,C 180,E1 9916.426,E2 9916.426} C_VEL
LIN {X 0,Y 341.597,Z 858.989,A -85,B 0,C 180,E1 9915.827,E2 9915.827} C_VEL
LIN {X 0,Y 354.414,Z 726.969,A -85,B 0,C 180,E1 9913.375,E2 9913.375} C_VEL
LIN {X 0,Y 351.541,Z 721.523,A -85,B 0,C 180,E1 9910.736,E2 9910.736} C_VEL
LIN {X 0,Y 350.158,Z 718.982,A -85,B 0,C 180,E1 9909.201,E2 9909.201} C_VEL
LIN {X 0,Y 348.419,Z 715.547,A -85,B 0,C 180,E1 9906.757,E2 9906.757} C_VEL
LIN {X 0,Y 346.626,Z 711.287,A -85,B 0,C 180,E1 9902.149,E2 9902.149} C_VEL
LIN {X 0,Y 346.683,Z 711.389,A -85,B 0,C 180,E1 9897.024,E2 9897.024} C_VEL
LIN {X 0,Y 348.479,Z 715.611,A -85,B 0,C 180,E1 9892.581,E2 9892.581} C_VEL
LIN {X 0,Y 351.244,Z 720.95,A -85,B 0,C 180,E1 9889.005,E2 9889.005} C_VEL
LIN {X 0,Y 354.042,Z 726.302,A -85,B 0,C 180,E1 9886.36,E2 9886.36} C_VEL
LIN {X 0,Y 354.277,Z 727.065,A -85,B 0,C 180,E1 9886.136,E2 9886.136} C_VEL
LIN {X 0,Y 339.765,Z 873.567,A -85,B 0,C 180,E1 9883.419,E2 9883.419} C_VEL
LIN {X 0,Y 335.834,Z 897.182,A -85,B 0,C 180,E1 9882.857,E2 9882.857} C_VEL
LIN {X 0,Y 331.13,Z 918.068,A -85,B 0,C 180,E1 9882.196,E2 9882.196} C_VEL
LIN {X 0,Y 325.062,Z 939.051,A -85,B 0,C 180,E1 9881.332,E2 9881.332} C_VEL
LIN {X 0,Y 317.694,Z 960.308,A -85,B 0,C 180,E1 9880.226,E2 9880.226} C_VEL
LIN {X 0,Y 309.215,Z 980.649,A -85,B 0,C 180,E1 9878.89,E2 9878.89} C_VEL
LIN {X 0,Y 299.747,Z 1000.578,A -85,B 0,C 180,E1 9877.268,E2 9877.268} C_VEL
LIN {X 0,Y 289.361,Z 1019.5,A -85,B 0,C 180,E1 9875.338,E2 9875.338} C_VEL
LIN {X 0,Y 277.858,Z 1038.303,A -85,B 0,C 180,E1 9872.953,E2 9872.953} C_VEL
LIN {X 0,Y 267.187,Z 1054.029,A -85,B 0,C 180,E1 9870.467,E2 9870.467} C_VEL
LIN {X 0,Y 255.219,Z 1070.201,A -85,B 0,C 180,E1 9867.273,E2 9867.273} C_VEL
LIN {X 0,Y 244.348,Z 1083.859,A -85,B 0,C 180,E1 9863.896,E2 9863.896} C_VEL
LIN {X 0,Y 233.13,Z 1097.056,A -85,B 0,C 180,E1 9859.767,E2 9859.767} C_VEL
LIN {X 0,Y 222.882,Z 1108.739,A -85,B 0,C 180,E1 9855.138,E2 9855.138} C_VEL
LIN {X 0,Y 213.504,Z 1119.039,A -85,B 0,C 180,E1 9849.822,E2 9849.822} C_VEL
LIN {X 0,Y 205.704,Z 1127.835,A -85,B 0,C 180,E1 9843.986,E2 9843.986} C_VEL
LIN {X 0,Y 199.945,Z 1134.596,A -85,B 0,C 180,E1 9838.039,E2 9838.039} C_VEL
LIN {X 0,Y 195.637,Z 1140.364,A -85,B 0,C 180,E1 9831.277,E2 9831.277} C_VEL
LIN {X 0,Y 193.339,Z 1144.1,A -85,B 0,C 180,E1 9824.986,E2 9824.986} C_VEL
LIN {X 0,Y 192.321,Z 1146.585,A -85,B 0,C 180,E1 9818.672,E2 9818.672} C_VEL
LIN {X 0,Y 192.054,Z 1147.6,A -85,B 0,C 180,E1 9812.985,E2 9812.985} C_VEL
LIN {X 0,Y 192.052,Z 1147.673,A -85,B 0,C 180,E1 9807.912,E2 9807.912} C_VEL
LIN {X 0,Y 192.201,Z 1146.931,A -85,B 0,C 180,E1 9802.828,E2 9802.828} C_VEL
LIN {X 0,Y 192.932,Z 1145.04,A -85,B 0,C 180,E1 9796.82,E2 9796.82} C_VEL
LIN {X 0,Y 194.922,Z 1141.435,A -85,B 0,C 180,E1 9790.212,E2 9790.212} C_VEL
LIN {X 0,Y 198.631,Z 1136.385,A -85,B 0,C 180,E1 9783.639,E2 9783.639} C_VEL
LIN {X 0,Y 204.099,Z 1129.685,A -85,B 0,C 180,E1 9777.393,E2 9777.393} C_VEL
LIN {X 0,Y 211.557,Z 1121.334,A -85,B 0,C 180,E1 9771.402,E2 9771.402} C_VEL
LIN {X 0,Y 220.41,Z 1111.474,A -85,B 0,C 180,E1 9766.048,E2 9766.048} C_VEL
LIN {X 0,Y 231.389,Z 1099.157,A -85,B 0,C 180,E1 9760.871,E2 9760.871} C_VEL
LIN {X 0,Y 242.15,Z 1086.64,A -85,B 0,C 180,E1 9756.771,E2 9756.771} C_VEL
LIN {X 0,Y 253.318,Z 1072.781,A -85,B 0,C 180,E1 9753.199,E2 9753.199} C_VEL
LIN {X 0,Y 264.651,Z 1057.819,A -85,B 0,C 180,E1 9750.099,E2 9750.099} C_VEL
LIN {X 0,Y 275.919,Z 1041.439,A -85,B 0,C 180,E1 9747.4,E2 9747.4} C_VEL
LIN {X 0,Y 286.983,Z 1023.936,A -85,B 0,C 180,E1 9745.062,E2 9745.062} C_VEL
LIN {X 0,Y 297.173,Z 1005.67,A -85,B 0,C 180,E1 9743.114,E2 9743.114} C_VEL
LIN {X 0,Y 306.716,Z 986.624,A -85,B 0,C 180,E1 9741.457,E2 9741.457} C_VEL
LIN {X 0,Y 315.136,Z 967.079,A -85,B 0,C 180,E1 9740.092,E2 9740.092} C_VEL
LIN {X 0,Y 322.896,Z 946.299,A -85,B 0,C 180,E1 9738.917,E2 9738.917} C_VEL
LIN {X 0,Y 329.083,Z 926.115,A -85,B 0,C 180,E1 9738.012,E2 9738.012} C_VEL
LIN {X 0,Y 334.781,Z 903.206,A -85,B 0,C 180,E1 9737.21,E2 9737.21} C_VEL
LIN {X 0,Y 338.835,Z 881.091,A -85,B 0,C 180,E1 9736.642,E2 9736.642} C_VEL
LIN {X 0,Y 342.43,Z 850.2,A -85,B 0,C 180,E1 9736.034,E2 9736.034} C_VEL
LIN {X 0,Y 347.441,Z 798.487,A -85,B 0,C 180,E1 9735.08,E2 9735.08} C_VEL
LIN {X 0,Y 347.931,Z 790.947,A -85,B 0,C 180,E1 9734.786,E2 9734.786} C_VEL
LIN {X 0,Y 348.363,Z 771.375,A -85,B 0,C 180,E1 9733.424,E2 9733.424} C_VEL
LIN {X 0,Y 348.844,Z 764.892,A -85,B 0,C 180,E1 9733.185,E2 9733.185} C_VEL
LIN {X 0,Y 352.079,Z 732.686,A -85,B 0,C 180,E1 9732.59,E2 9732.59} C_VEL
LIN {X 0,Y 349.299,Z 727.173,A -85,B 0,C 180,E1 9729.64,E2 9729.64} C_VEL
LIN {X 0,Y 347.434,Z 723.505,A -85,B 0,C 180,E1 9726.943,E2 9726.943} C_VEL
LIN {X 0,Y 345.805,Z 719.293,A -85,B 0,C 180,E1 9722.32,E2 9722.32} C_VEL
LIN {X 0,Y 345.856,Z 719.491,A -85,B 0,C 180,E1 9717.847,E2 9717.847} C_VEL
LIN {X 0,Y 347.638,Z 723.695,A -85,B 0,C 180,E1 9713.228,E2 9713.228} C_VEL
LIN {X 0,Y 350.192,Z 728.908,A -85,B 0,C 180,E1 9709.804,E2 9709.804} C_VEL
LIN {X 0,Y 352.194,Z 732.934,A -85,B 0,C 180,E1 9707.785,E2 9707.785} C_VEL
LIN {X 0,Y 337.276,Z 880.374,A -85,B 0,C 180,E1 9705.077,E2 9705.077} C_VEL
LIN {X 0,Y 333.191,Z 904.32,A -85,B 0,C 180,E1 9704.544,E2 9704.544} C_VEL
LIN {X 0,Y 328.074,Z 926.111,A -85,B 0,C 180,E1 9703.945,E2 9703.945} C_VEL
LIN {X 0,Y 321.717,Z 947.095,A -85,B 0,C 180,E1 9703.182,E2 9703.182} C_VEL
LIN {X 0,Y 314.022,Z 968.51,A -85,B 0,C 180,E1 9702.181,E2 9702.181} C_VEL
LIN {X 0,Y 305.073,Z 989.254,A -85,B 0,C 180,E1 9700.929,E2 9700.929} C_VEL
LIN {X 0,Y 295.302,Z 1009.192,A -85,B 0,C 180,E1 9699.422,E2 9699.422} C_VEL
LIN {X 0,Y 284.861,Z 1027.766,A -85,B 0,C 180,E1 9697.65,E2 9697.65} C_VEL
LIN {X 0,Y 272.834,Z 1047.035,A -85,B 0,C 180,E1 9695.346,E2 9695.346} C_VEL
LIN {X 0,Y 261.664,Z 1063.184,A -85,B 0,C 180,E1 9692.914,E2 9692.914} C_VEL
LIN {X 0,Y 248.956,Z 1080.069,A -85,B 0,C 180,E1 9689.709,E2 9689.709} C_VEL
LIN {X 0,Y 237.733,Z 1093.962,A -85,B 0,C 180,E1 9686.382,E2 9686.382} C_VEL
LIN {X 0,Y 225.623,Z 1108.06,A -85,B 0,C 180,E1 9682.074,E2 9682.074} C_VEL
LIN {X 0,Y 214.886,Z 1120.235,A -85,B 0,C 180,E1 9677.321,E2 9677.321} C_VEL
LIN {X 0,Y 204.977,Z 1131.171,A -85,B 0,C 180,E1 9671.729,E2 9671.729} C_VEL
LIN {X 0,Y 196.692,Z 1140.686,A -85,B 0,C 180,E1 9665.415,E2 9665.415} C_VEL
LIN {X 0,Y 190.912,Z 1147.846,A -85,B 0,C 180,E1 9659.147,E2 9659.147} C_VEL
LIN {X 0,Y 186.737,Z 1153.95,A -85,B 0,C 180,E1 9652.012,E2 9652.012} C_VEL
LIN {X 0,Y 184.785,Z 1157.815,A -85,B 0,C 180,E1 9645.696,E2 9645.696} C_VEL
LIN {X 0,Y 184.068,Z 1160.548,A -85,B 0,C 180,E1 9639.063,E2 9639.063} C_VEL
LIN {X 0,Y 184.016,Z 1161.689,A -85,B 0,C 180,E1 9633.114,E2 9633.114} C_VEL
LIN {X 0,Y 184.044,Z 1161.804,A -85,B 0,C 180,E1 9628.381,E2 9628.381} C_VEL
LIN {X 0,Y 184.012,Z 1161.124,A -85,B 0,C 180,E1 9623.447,E2 9623.447} C_VEL
LIN {X 0,Y 184.243,Z 1159.498,A -85,B 0,C 180,E1 9618.098,E2 9618.098} C_VEL
LIN {X 0,Y 185.494,Z 1156.283,A -85,B 0,C 180,E1 9611.456,E2 9611.456} C_VEL
LIN {X 0,Y 188.457,Z 1151.21,A -85,B 0,C 180,E1 9604.548,E2 9604.548} C_VEL
LIN {X 0,Y 193.418,Z 1144.652,A -85,B 0,C 180,E1 9597.828,E2 9597.828} C_VEL
LIN {X 0,Y 200.477,Z 1136.202,A -85,B 0,C 180,E1 9591.432,E2 9591.432} C_VEL
LIN {X 0,Y 209.593,Z 1125.992,A -85,B 0,C 180,E1 9585.47,E2 9585.47} C_VEL
LIN {X 0,Y 219.534,Z 1114.887,A -85,B 0,C 180,E1 9580.482,E2 9580.482} C_VEL
LIN {X 0,Y 231.513,Z 1101.172,A -85,B 0,C 180,E1 9575.713,E2 9575.713} C_VEL
LIN {X 0,Y 243.563,Z 1086.792,A -85,B 0,C 180,E1 9571.813,E2 9571.813} C_VEL
LIN {X 0,Y 255.905,Z 1070.841,A -85,B 0,C 180,E1 9568.463,E2 9568.463} C_VEL
LIN {X 0,Y 268.306,Z 1053.598,A -85,B 0,C 180,E1 9565.599,E2 9565.599} C_VEL
LIN {X 0,Y 278.977,Z 1037.235,A -85,B 0,C 180,E1 9563.434,E2 9563.434} C_VEL
LIN {X 0,Y 290.844,Z 1017.091,A -85,B 0,C 180,E1 9561.306,E2 9561.306} C_VEL
LIN {X 0,Y 300.205,Z 999.187,A -85,B 0,C 180,E1 9559.796,E2 9559.796} C_VEL
LIN {X 0,Y 309.781,Z 978.318,A -85,B 0,C 180,E1 9558.389,E2 9558.389} C_VEL
LIN {X 0,Y 317.716,Z 958.213,A -85,B 0,C 180,E1 9557.315,E2 9557.315} C_VEL
LIN {X 0,Y 325.155,Z 935.577,A -85,B 0,C 180,E1 9556.379,E2 9556.379} C_VEL
LIN {X 0,Y 331.245,Z 912.785,A -85,B 0,C 180,E1 9555.674,E2 9555.674} C_VEL
LIN {X 0,Y 335.742,Z 889.455,A -85,B 0,C 180,E1 9555.123,E2 9555.123} C_VEL
LIN {X 0,Y 339.125,Z 862.378,A -85,B 0,C 180,E1 9554.588,E2 9554.588} C_VEL
LIN {X 0,Y 352.012,Z 732.771,A -85,B 0,C 180,E1 9552.208,E2 9552.208} C_VEL
LIN {X 0,Y 349.385,Z 727.43,A -85,B 0,C 180,E1 9549.471,E2 9549.471} C_VEL
LIN {X 0,Y 347.337,Z 723.425,A -85,B 0,C 180,E1 9546.612,E2 9546.612} C_VEL
LIN {X 0,Y 345.613,Z 719.213,A -85,B 0,C 180,E1 9541.989,E2 9541.989} C_VEL
LIN {X 0,Y 345.669,Z 719.286,A -85,B 0,C 180,E1 9537.181,E2 9537.181} C_VEL
LIN {X 0,Y 347.397,Z 723.49,A -85,B 0,C 180,E1 9532.724,E2 9532.724} C_VEL
LIN {X 0,Y 349.949,Z 728.652,A -85,B 0,C 180,E1 9529.297,E2 9529.297} C_VEL
LIN {X 0,Y 351.92,Z 732.572,A -85,B 0,C 180,E1 9527.305,E2 9527.305} C_VEL
LIN {X 0,Y 337.556,Z 873.995,A -85,B 0,C 180,E1 9524.719,E2 9524.719} C_VEL
LIN {X 0,Y 333.548,Z 897.566,A -85,B 0,C 180,E1 9524.17,E2 9524.17} C_VEL
LIN {X 0,Y 328.661,Z 918.812,A -85,B 0,C 180,E1 9523.512,E2 9523.512} C_VEL
LIN {X 0,Y 322.16,Z 940.638,A -85,B 0,C 180,E1 9522.626,E2 9522.626} C_VEL
LIN {X 0,Y 314.647,Z 961.714,A -85,B 0,C 180,E1 9521.543,E2 9521.543} C_VEL
LIN {X 0,Y 305.99,Z 981.851,A -85,B 0,C 180,E1 9520.235,E2 9520.235} C_VEL
LIN {X 0,Y 296.107,Z 1001.98,A -85,B 0,C 180,E1 9518.612,E2 9518.612} C_VEL
LIN {X 0,Y 285.675,Z 1020.471,A -85,B 0,C 180,E1 9516.746,E2 9516.746} C_VEL
LIN {X 0,Y 273.418,Z 1039.817,A -85,B 0,C 180,E1 9514.3,E2 9514.3} C_VEL
LIN {X 0,Y 262.176,Z 1055.84,A -85,B 0,C 180,E1 9511.761,E2 9511.761} C_VEL
LIN {X 0,Y 250.375,Z 1071.12,A -85,B 0,C 180,E1 9508.717,E2 9508.717} C_VEL
LIN {X 0,Y 238.679,Z 1085.266,A -85,B 0,C 180,E1 9505.194,E2 9505.194} C_VEL
LIN {X 0,Y 227.309,Z 1097.99,A -85,B 0,C 180,E1 9501.131,E2 9501.131} C_VEL
LIN {X 0,Y 216.62,Z 1109.586,A -85,B 0,C 180,E1 9496.442,E2 9496.442} C_VEL
LIN {X 0,Y 206.837,Z 1119.75,A -85,B 0,C 180,E1 9491.051,E2 9491.051} C_VEL
LIN {X 0,Y 198.123,Z 1128.945,A -85,B 0,C 180,E1 9484.653,E2 9484.653} C_VEL
LIN {X 0,Y 192.046,Z 1135.705,A -85,B 0,C 180,E1 9478.372,E2 9478.372} C_VEL
LIN {X 0,Y 187.57,Z 1141.265,A -85,B 0,C 180,E1 9471.253,E2 9471.253} C_VEL
LIN {X 0,Y 185.268,Z 1144.863,A -85,B 0,C 180,E1 9464.694,E2 9464.694} C_VEL
LIN {X 0,Y 184.269,Z 1147.078,A -85,B 0,C 180,E1 9458.111,E2 9458.111} C_VEL
LIN {X 0,Y 184.059,Z 1147.921,A -85,B 0,C 180,E1 9452.803,E2 9452.803} C_VEL
LIN {X 0,Y 184.059,Z 1147.973,A -85,B 0,C 180,E1 9447.821,E2 9447.821} C_VEL
LIN {X 0,Y 184.224,Z 1147.232,A -85,B 0,C 180,E1 9442.516,E2 9442.516} C_VEL
LIN {X 0,Y 185.046,Z 1145.344,A -85,B 0,C 180,E1 9436.247,E2 9436.247} C_VEL
LIN {X 0,Y 187.249,Z 1141.741,A -85,B 0,C 180,E1 9429.365,E2 9429.365} C_VEL
LIN {X 0,Y 191.237,Z 1136.744,A -85,B 0,C 180,E1 9422.607,E2 9422.607} C_VEL
LIN {X 0,Y 197.184,Z 1129.994,A -85,B 0,C 180,E1 9416.098,E2 9416.098} C_VEL
LIN {X 0,Y 205.258,Z 1121.525,A -85,B 0,C 180,E1 9409.888,E2 9409.888} C_VEL
LIN {X 0,Y 214.527,Z 1111.783,A -85,B 0,C 180,E1 9404.513,E2 9404.513} C_VEL
LIN {X 0,Y 226.322,Z 1099.178,A -85,B 0,C 180,E1 9399.18,E2 9399.18} C_VEL
LIN {X 0,Y 237.93,Z 1086.259,A -85,B 0,C 180,E1 9394.97,E2 9394.97} C_VEL
LIN {X 0,Y 249.847,Z 1071.919,A -85,B 0,C 180,E1 9391.349,E2 9391.349} C_VEL
LIN {X 0,Y 262.051,Z 1056.196,A -85,B 0,C 180,E1 9388.19,E2 9388.19} C_VEL
LIN {X 0,Y 273.366,Z 1040.097,A -85,B 0,C 180,E1 9385.632,E2 9385.632} C_VEL
LIN {X 0,Y 285.55,Z 1020.935,A -85,B 0,C 180,E1 9383.199,E2 9383.199} C_VEL
LIN {X 0,Y 295.974,Z 1002.507,A -85,B 0,C 180,E1 9381.333,E2 9381.333} C_VEL
LIN {X 0,Y 305.873,Z 982.455,A -85,B 0,C 180,E1 9379.706,E2 9379.706} C_VEL
LIN {X 0,Y 314.531,Z 962.385,A -85,B 0,C 180,E1 9378.396,E2 9378.396} C_VEL
LIN {X 0,Y 322.149,Z 941.175,A -85,B 0,C 180,E1 9377.299,E2 9377.299} C_VEL
LIN {X 0,Y 328.645,Z 919.578,A -85,B 0,C 180,E1 9376.415,E2 9376.415} C_VEL
LIN {X 0,Y 333.627,Z 898.011,A -85,B 0,C 180,E1 9375.744,E2 9375.744} C_VEL
LIN {X 0,Y 337.65,Z 874.653,A -85,B 0,C 180,E1 9375.196,E2 9375.196} C_VEL
LIN {X 0,Y 347.711,Z 776.141,A -85,B 0,C 180,E1 9373.388,E2 9373.388} C_VEL
LIN {X 0,Y 348.844,Z 764.892,A -85,B 0,C 180,E1 9373.185,E2 9373.185} C_VEL
LIN {X 0,Y 349.122,Z 759.896,A -85,B 0,C 180,E1 9372.933,E2 9372.933} C_VEL
LIN {X 0,Y 349.081,Z 747.5,A -85,B 0,C 180,E1 9371.707,E2 9371.707} C_VEL
LIN {X 0,Y 349.375,Z 743.188,A -85,B 0,C 180,E1 9371.506,E2 9371.506} C_VEL
LIN {X 0,Y 349.851,Z 738.503,A -85,B 0,C 180,E1 9371.415,E2 9371.415} C_VEL
LIN {X 0,Y 347.851,Z 734.544,A -85,B 0,C 180,E1 9369.096,E2 9369.096} C_VEL
LIN {X 0,Y 346.358,Z 731.384,A -85,B 0,C 180,E1 9366.798,E2 9366.798} C_VEL
LIN {X 0,Y 344.798,Z 727.219,A -85,B 0,C 180,E1 9362.161,E2 9362.161} C_VEL
LIN {X 0,Y 344.847,Z 727.382,A -85,B 0,C 180,E1 9358.006,E2 9358.006} C_VEL
LIN {X 0,Y 346.736,Z 732.115,A -85,B 0,C 180,E1 9353.044,E2 9353.044} C_VEL
LIN {X 0,Y 348.904,Z 736.605,A -85,B 0,C 180,E1 9350.1,E2 9350.1} C_VEL
LIN {X 0,Y 349.941,Z 738.833,A -85,B 0,C 180,E1 9348.959,E2 9348.959} C_VEL
LIN {X 0,Y 335.292,Z 880.115,A -85,B 0,C 180,E1 9346.405,E2 9346.405} C_VEL
LIN {X 0,Y 331.132,Z 904.055,A -85,B 0,C 180,E1 9345.885,E2 9345.885} C_VEL
LIN {X 0,Y 325.651,Z 926.896,A -85,B 0,C 180,E1 9345.275,E2 9345.275} C_VEL
LIN {X 0,Y 319.033,Z 948.09,A -85,B 0,C 180,E1 9344.518,E2 9344.518} C_VEL
LIN {X 0,Y 311.244,Z 969.165,A -85,B 0,C 180,E1 9343.552,E2 9343.552} C_VEL
LIN {X 0,Y 302.194,Z 989.623,A -85,B 0,C 180,E1 9342.344,E2 9342.344} C_VEL
LIN {X 0,Y 291.596,Z 1010.541,A -85,B 0,C 180,E1 9340.782,E2 9340.782} C_VEL
LIN {X 0,Y 280.892,Z 1029.036,A -85,B 0,C 180,E1 9339.034,E2 9339.034} C_VEL
LIN {X 0,Y 268.508,Z 1048.14,A -85,B 0,C 180,E1 9336.752,E2 9336.752} C_VEL
LIN {X 0,Y 256.499,Z 1064.93,A -85,B 0,C 180,E1 9334.219,E2 9334.219} C_VEL
LIN {X 0,Y 244.151,Z 1080.618,A -85,B 0,C 180,E1 9331.209,E2 9331.209} C_VEL
LIN {X 0,Y 231.888,Z 1095.225,A -85,B 0,C 180,E1 9327.68,E2 9327.68} C_VEL
LIN {X 0,Y 219.401,Z 1109.016,A -85,B 0,C 180,E1 9323.346,E2 9323.346} C_VEL
LIN {X 0,Y 207.713,Z 1121.523,A -85,B 0,C 180,E1 9318.255,E2 9318.255} C_VEL
LIN {X 0,Y 198.152,Z 1131.543,A -85,B 0,C 180,E1 9312.937,E2 9312.937} C_VEL
LIN {X 0,Y 189.248,Z 1141.103,A -85,B 0,C 180,E1 9306.279,E2 9306.279} C_VEL
LIN {X 0,Y 183.189,Z 1148.162,A -85,B 0,C 180,E1 9299.78,E2 9299.78} C_VEL
LIN {X 0,Y 178.81,Z 1154.073,A -85,B 0,C 180,E1 9292.348,E2 9292.348} C_VEL
LIN {X 0,Y 176.781,Z 1157.845,A -85,B 0,C 180,E1 9285.752,E2 9285.752} C_VEL
LIN {X 0,Y 176.063,Z 1160.393,A -85,B 0,C 180,E1 9278.819,E2 9278.819} C_VEL
LIN {X 0,Y 176.02,Z 1161.389,A -85,B 0,C 180,E1 9273.256,E2 9273.256} C_VEL
LIN {X 0,Y 176.049,Z 1161.504,A -85,B 0,C 180,E1 9268.308,E2 9268.308} C_VEL
LIN {X 0,Y 176.011,Z 1160.822,A -85,B 0,C 180,E1 9263.148,E2 9263.148} C_VEL
LIN {X 0,Y 176.296,Z 1159.193,A -85,B 0,C 180,E1 9257.553,E2 9257.553} C_VEL
LIN {X 0,Y 177.826,Z 1155.777,A -85,B 0,C 180,E1 9250.283,E2 9250.283} C_VEL
LIN {X 0,Y 180.991,Z 1150.898,A -85,B 0,C 180,E1 9243.417,E2 9243.417} C_VEL
LIN {X 0,Y 186.402,Z 1144.338,A -85,B 0,C 180,E1 9236.461,E2 9236.461} C_VEL
LIN {X 0,Y 193.991,Z 1135.886,A -85,B 0,C 180,E1 9229.888,E2 9229.888} C_VEL
LIN {X 0,Y 203.733,Z 1125.624,A -85,B 0,C 180,E1 9223.786,E2 9223.786} C_VEL
LIN {X 0,Y 214.183,Z 1114.57,A -85,B 0,C 180,E1 9218.775,E2 9218.775} C_VEL
LIN {X 0,Y 226.723,Z 1100.855,A -85,B 0,C 180,E1 9213.993,E2 9213.993} C_VEL
LIN {X 0,Y 239.4,Z 1086.322,A -85,B 0,C 180,E1 9210.077,E2 9210.077} C_VEL
LIN {X 0,Y 252.052,Z 1070.527,A -85,B 0,C 180,E1 9206.803,E2 9206.803} C_VEL
LIN {X 0,Y 264.835,Z 1053.284,A -85,B 0,C 180,E1 9203.984,E2 9203.984} C_VEL
LIN {X 0,Y 275.804,Z 1036.922,A -85,B 0,C 180,E1 9201.863,E2 9201.863} C_VEL
LIN {X 0,Y 287.966,Z 1016.779,A -85,B 0,C 180,E1 9199.786,E2 9199.786} C_VEL
LIN {X 0,Y 297.5,Z 998.953,A -85,B 0,C 180,E1 9198.322,E2 9198.322} C_VEL
LIN {X 0,Y 307.314,Z 978.007,A -85,B 0,C 180,E1 9196.951,E2 9196.951} C_VEL
LIN {X 0,Y 315.088,Z 958.713,A -85,B 0,C 180,E1 9195.948,E2 9195.948} C_VEL
LIN {X 0,Y 322.751,Z 936.008,A -85,B 0,C 180,E1 9195.03,E2 9195.03} C_VEL
LIN {X 0,Y 328.831,Z 913.767,A -85,B 0,C 180,E1 9194.359,E2 9194.359} C_VEL
LIN {X 0,Y 333.515,Z 890.44,A -85,B 0,C 180,E1 9193.816,E2 9193.816} C_VEL
LIN {X 0,Y 336.789,Z 866.008,A -85,B 0,C 180,E1 9193.335,E2 9193.335} C_VEL
LIN {X 0,Y 349.784,Z 738.511,A -85,B 0,C 180,E1 9191.041,E2 9191.041} C_VEL
LIN {X 0,Y 347.717,Z 734.476,A -85,B 0,C 180,E1 9188.682,E2 9188.682} C_VEL
LIN {X 0,Y 346.156,Z 731.178,A -85,B 0,C 180,E1 9186.301,E2 9186.301} C_VEL
LIN {X 0,Y 344.601,Z 727.14,A -85,B 0,C 180,E1 9181.829,E2 9181.829} C_VEL
LIN {X 0,Y 344.677,Z 727.371,A -85,B 0,C 180,E1 9177.173,E2 9177.173} C_VEL
LIN {X 0,Y 346.551,Z 731.963,A -85,B 0,C 180,E1 9172.456,E2 9172.456} C_VEL
LIN {X 0,Y 348.732,Z 736.508,A -85,B 0,C 180,E1 9169.51,E2 9169.51} C_VEL
LIN {X 0,Y 349.655,Z 738.638,A -85,B 0,C 180,E1 9168.479,E2 9168.479} C_VEL
LIN {X 0,Y 335.537,Z 874.317,A -85,B 0,C 180,E1 9166.037,E2 9166.037} C_VEL
LIN {X 0,Y 331.472,Z 897.787,A -85,B 0,C 180,E1 9165.504,E2 9165.504} C_VEL
LIN {X 0,Y 326.503,Z 919.016,A -85,B 0,C 180,E1 9164.866,E2 9164.866} C_VEL
LIN {X 0,Y 319.894,Z 940.82,A -85,B 0,C 180,E1 9164.006,E2 9164.006} C_VEL
LIN {X 0,Y 312.19,Z 962.023,A -85,B 0,C 180,E1 9162.946,E2 9162.946} C_VEL
LIN {X 0,Y 303.353,Z 982.16,A -85,B 0,C 180,E1 9161.671,E2 9161.671} C_VEL
LIN {X 0,Y 293.454,Z 1001.923,A -85,B 0,C 180,E1 9160.119,E2 9160.119} C_VEL
LIN {X 0,Y 282.959,Z 1020.119,A -85,B 0,C 180,E1 9158.333,E2 9158.333} C_VEL
LIN {X 0,Y 270.887,Z 1038.83,A -85,B 0,C 180,E1 9156.045,E2 9156.045} C_VEL
LIN {X 0,Y 259.499,Z 1054.651,A -85,B 0,C 180,E1 9153.617,E2 9153.617} C_VEL
LIN {X 0,Y 246.902,Z 1070.599,A -85,B 0,C 180,E1 9150.538,E2 9150.538} C_VEL
LIN {X 0,Y 235.371,Z 1084.063,A -85,B 0,C 180,E1 9147.259,E2 9147.259} C_VEL
LIN {X 0,Y 222.817,Z 1097.68,A -85,B 0,C 180,E1 9143.012,E2 9143.012} C_VEL
LIN {X 0,Y 211.526,Z 1109.364,A -85,B 0,C 180,E1 9138.319,E2 9138.319} C_VEL
LIN {X 0,Y 201.184,Z 1119.549,A -85,B 0,C 180,E1 9132.913,E2 9132.913} C_VEL
LIN {X 0,Y 192.228,Z 1128.457,A -85,B 0,C 180,E1 9126.74,E2 9126.74} C_VEL
LIN {X 0,Y 185.571,Z 1135.215,A -85,B 0,C 180,E1 9120.43,E2 9120.43} C_VEL
LIN {X 0,Y 180.293,Z 1141.177,A -85,B 0,C 180,E1 9112.844,E2 9112.844} C_VEL
LIN {X 0,Y 177.679,Z 1144.711,A -85,B 0,C 180,E1 9106.343,E2 9106.343} C_VEL
LIN {X 0,Y 176.383,Z 1147.252,A -85,B 0,C 180,E1 9099.134,E2 9099.134} C_VEL
LIN {X 0,Y 176.066,Z 1148.222,A -85,B 0,C 180,E1 9092.93,E2 9092.93} C_VEL
LIN {X 0,Y 176.064,Z 1148.272,A -85,B 0,C 180,E1 9087.722,E2 9087.722} C_VEL
LIN {X 0,Y 176.249,Z 1147.534,A -85,B 0,C 180,E1 9082.175,E2 9082.175} C_VEL
LIN {X 0,Y 177.174,Z 1145.648,A -85,B 0,C 180,E1 9075.623,E2 9075.623} C_VEL
LIN {X 0,Y 179.665,Z 1141.982,A -85,B 0,C 180,E1 9068.339,E2 9068.339} C_VEL
LIN {X 0,Y 184.207,Z 1136.794,A -85,B 0,C 180,E1 9061.114,E2 9061.114} C_VEL
LIN {X 0,Y 190.723,Z 1129.961,A -85,B 0,C 180,E1 9054.415,E2 9054.415} C_VEL
LIN {X 0,Y 199.314,Z 1121.505,A -85,B 0,C 180,E1 9048.15,E2 9048.15} C_VEL
LIN {X 0,Y 209.029,Z 1111.875,A -85,B 0,C 180,E1 9042.785,E2 9042.785} C_VEL
LIN {X 0,Y 220.92,Z 1099.774,A -85,B 0,C 180,E1 9037.625,E2 9037.625} C_VEL
LIN {X 0,Y 232.651,Z 1087.254,A -85,B 0,C 180,E1 9033.515,E2 9033.515} C_VEL
LIN {X 0,Y 245.206,Z 1072.776,A -85,B 0,C 180,E1 9029.833,E2 9029.833} C_VEL
LIN {X 0,Y 257.546,Z 1057.498,A -85,B 0,C 180,E1 9026.758,E2 9026.758} C_VEL
LIN {X 0,Y 269.548,Z 1040.948,A -85,B 0,C 180,E1 9024.146,E2 9024.146} C_VEL
LIN {X 0,Y 281.256,Z 1023.219,A -85,B 0,C 180,E1 9021.898,E2 9021.898} C_VEL
LIN {X 0,Y 291.705,Z 1005.332,A -85,B 0,C 180,E1 9020.087,E2 9020.087} C_VEL
LIN {X 0,Y 302.411,Z 984.539,A -85,B 0,C 180,E1 9018.395,E2 9018.395} C_VEL
LIN {X 0,Y 311.232,Z 964.677,A -85,B 0,C 180,E1 9017.11,E2 9017.11} C_VEL
LIN {X 0,Y 319.34,Z 942.998,A -85,B 0,C 180,E1 9015.994,E2 9015.994} C_VEL
LIN {X 0,Y 325.586,Z 922.941,A -85,B 0,C 180,E1 9015.177,E2 9015.177} C_VEL
LIN {X 0,Y 331.136,Z 900.246,A -85,B 0,C 180,E1 9014.463,E2 9014.463} C_VEL
LIN {X 0,Y 335.31,Z 877.449,A -85,B 0,C 180,E1 9013.927,E2 9013.927} C_VEL
LIN {X 0,Y 340.503,Z 829.608,A -85,B 0,C 180,E1 9013.048,E2 9013.048} C_VEL
LIN {X 0,Y 349.375,Z 743.188,A -85,B 0,C 180,E1 9011.506,E2 9011.506} C_VEL
LIN {X 0,Y 349.377,Z 741.187,A -85,B 0,C 180,E1 9011.3,E2 9011.3} C_VEL
LIN {X 0,Y 348.979,Z 739.858,A -85,B 0,C 180,E1 9010.815,E2 9010.815} C_VEL
LIN {X 0,Y 348.114,Z 739.629,A -85,B 0,C 180,E1 9009.996,E2 9009.996} C_VEL
LIN {X 0,Y 346.258,Z 740.985,A -85,B 0,C 180,E1 9008.21,E2 9008.21} C_VEL
LIN {X 0,Y 345.828,Z 740.56,A -85,B 0,C 180,E1 9007.617,E2 9007.617} C_VEL
LIN {X 0,Y 345.19,Z 739.139,A -85,B 0,C 180,E1 9006.487,E2 9006.487} C_VEL
LIN {X 0,Y 343.793,Z 735.146,A -85,B 0,C 180,E1 9002,E2 9002} C_VEL
LIN {X 0,Y 343.841,Z 735.273,A -85,B 0,C 180,E1 8998.167,E2 8998.167} C_VEL
LIN {X 0,Y 345.597,Z 739.933,A -85,B 0,C 180,E1 8993.272,E2 8993.272} C_VEL
LIN {X 0,Y 347.693,Z 744.452,A -85,B 0,C 180,E1 8990.316,E2 8990.316} C_VEL
LIN {X 0,Y 347.805,Z 745.011,A -85,B 0,C 180,E1 8990.146,E2 8990.146} C_VEL
LIN {X 0,Y 333.481,Z 879.92,A -85,B 0,C 180,E1 8987.747,E2 8987.747} C_VEL
LIN {X 0,Y 329.24,Z 903.866,A -85,B 0,C 180,E1 8987.241,E2 8987.241} C_VEL
LIN {X 0,Y 323.696,Z 926.604,A -85,B 0,C 180,E1 8986.654,E2 8986.654} C_VEL
LIN {X 0,Y 317.013,Z 947.666,A -85,B 0,C 180,E1 8985.933,E2 8985.933} C_VEL
LIN {X 0,Y 309.09,Z 968.758,A -85,B 0,C 180,E1 8985.002,E2 8985.002} C_VEL
LIN {X 0,Y 299.821,Z 989.323,A -85,B 0,C 180,E1 8983.829,E2 8983.829} C_VEL
LIN {X 0,Y 289.101,Z 1010.069,A -85,B 0,C 180,E1 8982.33,E2 8982.33} C_VEL
LIN {X 0,Y 278.194,Z 1028.506,A -85,B 0,C 180,E1 8980.639,E2 8980.639} C_VEL
LIN {X 0,Y 265.159,Z 1048.106,A -85,B 0,C 180,E1 8978.356,E2 8978.356} C_VEL
LIN {X 0,Y 252.589,Z 1065.17,A -85,B 0,C 180,E1 8975.823,E2 8975.823} C_VEL
LIN {X 0,Y 239.519,Z 1081.166,A -85,B 0,C 180,E1 8972.767,E2 8972.767} C_VEL
LIN {X 0,Y 226.831,Z 1095.678,A -85,B 0,C 180,E1 8969.249,E2 8969.249} C_VEL
LIN {X 0,Y 214.477,Z 1108.731,A -85,B 0,C 180,E1 8965.133,E2 8965.133} C_VEL
LIN {X 0,Y 202.093,Z 1121.33,A -85,B 0,C 180,E1 8959.972,E2 8959.972} C_VEL
LIN {X 0,Y 191.631,Z 1131.701,A -85,B 0,C 180,E1 8954.359,E2 8954.359} C_VEL
LIN {X 0,Y 182.205,Z 1141.155,A -85,B 0,C 180,E1 8947.525,E2 8947.525} C_VEL
LIN {X 0,Y 175.49,Z 1148.479,A -85,B 0,C 180,E1 8940.469,E2 8940.469} C_VEL
LIN {X 0,Y 171.042,Z 1153.981,A -85,B 0,C 180,E1 8933.057,E2 8933.057} C_VEL
LIN {X 0,Y 168.776,Z 1157.874,A -85,B 0,C 180,E1 8925.813,E2 8925.813} C_VEL
LIN {X 0,Y 168.059,Z 1160.237,A -85,B 0,C 180,E1 8918.553,E2 8918.553} C_VEL
LIN {X 0,Y 168.027,Z 1161.113,A -85,B 0,C 180,E1 8913.069,E2 8913.069} C_VEL
LIN {X 0,Y 168.047,Z 1161.184,A -85,B 0,C 180,E1 8907.953,E2 8907.953} C_VEL
LIN {X 0,Y 168.016,Z 1160.447,A -85,B 0,C 180,E1 8902.476,E2 8902.476} C_VEL
LIN {X 0,Y 168.441,Z 1158.645,A -85,B 0,C 180,E1 8896.264,E2 8896.264} C_VEL
LIN {X 0,Y 170.466,Z 1154.819,A -85,B 0,C 180,E1 8888.313,E2 8888.313} C_VEL
LIN {X 0,Y 174.056,Z 1150.045,A -85,B 0,C 180,E1 8881.508,E2 8881.508} C_VEL
LIN {X 0,Y 180.812,Z 1142.566,A -85,B 0,C 180,E1 8873.722,E2 8873.722} C_VEL
LIN {X 0,Y 188.963,Z 1134.3,A -85,B 0,C 180,E1 8867.347,E2 8867.347} C_VEL
LIN {X 0,Y 199.525,Z 1123.777,A -85,B 0,C 180,E1 8861.263,E2 8861.263} C_VEL
LIN {X 0,Y 210.818,Z 1112.495,A -85,B 0,C 180,E1 8856.265,E2 8856.265} C_VEL
LIN {X 0,Y 222.912,Z 1099.715,A -85,B 0,C 180,E1 8851.956,E2 8851.956} C_VEL
LIN {X 0,Y 235.909,Z 1085.321,A -85,B 0,C 180,E1 8848.166,E2 8848.166} C_VEL
LIN {X 0,Y 248.795,Z 1069.743,A -85,B 0,C 180,E1 8845.007,E2 8845.007} C_VEL
LIN {X 0,Y 262.433,Z 1051.755,A -85,B 0,C 180,E1 8842.159,E2 8842.159} C_VEL
LIN {X 0,Y 273.662,Z 1035.38,A -85,B 0,C 180,E1 8840.116,E2 8840.116} C_VEL
LIN {X 0,Y 285.982,Z 1015.251,A -85,B 0,C 180,E1 8838.129,E2 8838.129} C_VEL
LIN {X 0,Y 296.009,Z 996.795,A -85,B 0,C 180,E1 8836.685,E2 8836.685} C_VEL
LIN {X 0,Y 305.48,Z 976.685,A -85,B 0,C 180,E1 8835.435,E2 8835.435} C_VEL
LIN {X 0,Y 313.852,Z 956.13,A -85,B 0,C 180,E1 8834.422,E2 8834.422} C_VEL
LIN {X 0,Y 321.203,Z 934.211,A -85,B 0,C 180,E1 8833.59,E2 8833.59} C_VEL
LIN {X 0,Y 327.433,Z 911.428,A -85,B 0,C 180,E1 8832.942,E2 8832.942} C_VEL
LIN {X 0,Y 331.989,Z 888.33,A -85,B 0,C 180,E1 8832.429,E2 8832.429} C_VEL
LIN {X 0,Y 335.726,Z 858.861,A -85,B 0,C 180,E1 8831.874,E2 8831.874} C_VEL
LIN {X 0,Y 347.62,Z 744.539,A -85,B 0,C 180,E1 8829.816,E2 8829.816} C_VEL
LIN {X 0,Y 346.064,Z 741.366,A -85,B 0,C 180,E1 8827.804,E2 8827.804} C_VEL
LIN {X 0,Y 344.986,Z 738.929,A -85,B 0,C 180,E1 8825.989,E2 8825.989} C_VEL
LIN {X 0,Y 343.593,Z 735.068,A -85,B 0,C 180,E1 8821.667,E2 8821.667} C_VEL
LIN {X 0,Y 343.666,Z 735.266,A -85,B 0,C 180,E1 8817.332,E2 8817.332} C_VEL
LIN {X 0,Y 345.412,Z 739.785,A -85,B 0,C 180,E1 8812.682,E2 8812.682} C_VEL
LIN {X 0,Y 347.46,Z 744.223,A -85,B 0,C 180,E1 8809.798,E2 8809.798} C_VEL
LIN {X 0,Y 347.53,Z 744.778,A -85,B 0,C 180,E1 8809.667,E2 8809.667} C_VEL
LIN {X 0,Y 333.697,Z 874.639,A -85,B 0,C 180,E1 8807.37,E2 8807.37} C_VEL
LIN {X 0,Y 329.54,Z 898.193,A -85,B 0,C 180,E1 8806.849,E2 8806.849} C_VEL
LIN {X 0,Y 324.392,Z 919.76,A -85,B 0,C 180,E1 8806.219,E2 8806.219} C_VEL
LIN {X 0,Y 317.773,Z 941.129,A -85,B 0,C 180,E1 8805.399,E2 8805.399} C_VEL
LIN {X 0,Y 309.923,Z 962.331,A -85,B 0,C 180,E1 8804.37,E2 8804.37} C_VEL
LIN {X 0,Y 300.91,Z 982.468,A -85,B 0,C 180,E1 8803.132,E2 8803.132} C_VEL
LIN {X 0,Y 290.799,Z 1002.232,A -85,B 0,C 180,E1 8801.621,E2 8801.621} C_VEL
LIN {X 0,Y 280.06,Z 1020.428,A -85,B 0,C 180,E1 8799.878,E2 8799.878} C_VEL
LIN {X 0,Y 268.007,Z 1038.684,A -85,B 0,C 180,E1 8797.704,E2 8797.704} C_VEL
LIN {X 0,Y 256.26,Z 1054.574,A -85,B 0,C 180,E1 8795.324,E2 8795.324} C_VEL
LIN {X 0,Y 242.964,Z 1070.911,A -85,B 0,C 180,E1 8792.226,E2 8792.226} C_VEL
LIN {X 0,Y 231.015,Z 1084.375,A -85,B 0,C 180,E1 8788.979,E2 8788.979} C_VEL
LIN {X 0,Y 217.948,Z 1097.992,A -85,B 0,C 180,E1 8784.747,E2 8784.747} C_VEL
LIN {X 0,Y 206.114,Z 1109.677,A -85,B 0,C 180,E1 8780.038,E2 8780.038} C_VEL
LIN {X 0,Y 195.203,Z 1119.861,A -85,B 0,C 180,E1 8774.567,E2 8774.567} C_VEL
LIN {X 0,Y 185.669,Z 1128.768,A -85,B 0,C 180,E1 8768.266,E2 8768.266} C_VEL
LIN {X 0,Y 178.287,Z 1135.753,A -85,B 0,C 180,E1 8761.521,E2 8761.521} C_VEL
LIN {X 0,Y 172.584,Z 1141.683,A -85,B 0,C 180,E1 8753.563,E2 8753.563} C_VEL
LIN {X 0,Y 169.785,Z 1145.169,A -85,B 0,C 180,E1 8746.773,E2 8746.773} C_VEL
LIN {X 0,Y 168.395,Z 1147.618,A -85,B 0,C 180,E1 8739.226,E2 8739.226} C_VEL
LIN {X 0,Y 168.072,Z 1148.522,A -85,B 0,C 180,E1 8733.07,E2 8733.07} C_VEL
LIN {X 0,Y 168.07,Z 1148.572,A -85,B 0,C 180,E1 8727.614,E2 8727.614} C_VEL
LIN {X 0,Y 168.258,Z 1147.899,A -85,B 0,C 180,E1 8722.145,E2 8722.145} C_VEL
LIN {X 0,Y 169.165,Z 1146.166,A -85,B 0,C 180,E1 8715.627,E2 8715.627} C_VEL
LIN {X 0,Y 171.862,Z 1142.551,A -85,B 0,C 180,E1 8707.781,E2 8707.781} C_VEL
LIN {X 0,Y 176.248,Z 1137.849,A -85,B 0,C 180,E1 8700.799,E2 8700.799} C_VEL
LIN {X 0,Y 183.333,Z 1130.954,A -85,B 0,C 180,E1 8693.526,E2 8693.526} C_VEL
LIN {X 0,Y 192.313,Z 1122.702,A -85,B 0,C 180,E1 8687.072,E2 8687.072} C_VEL
LIN {X 0,Y 203.021,Z 1112.624,A -85,B 0,C 180,E1 8681.296,E2 8681.296} C_VEL
LIN {X 0,Y 215.361,Z 1100.704,A -85,B 0,C 180,E1 8676.116,E2 8676.116} C_VEL
LIN {X 0,Y 227.529,Z 1088.249,A -85,B 0,C 180,E1 8671.992,E2 8671.992} C_VEL
LIN {X 0,Y 240.747,Z 1073.629,A -85,B 0,C 180,E1 8668.26,E2 8668.26} C_VEL
LIN {X 0,Y 253.454,Z 1058.43,A -85,B 0,C 180,E1 8665.218,E2 8665.218} C_VEL
LIN {X 0,Y 265.917,Z 1041.799,A -85,B 0,C 180,E1 8662.618,E2 8662.618} C_VEL
LIN {X 0,Y 277.814,Z 1024.35,A -85,B 0,C 180,E1 8660.433,E2 8660.433} C_VEL
LIN {X 0,Y 289.018,Z 1005.632,A -85,B 0,C 180,E1 8658.576,E2 8658.576} C_VEL
LIN {X 0,Y 299.958,Z 984.837,A -85,B 0,C 180,E1 8656.929,E2 8656.929} C_VEL
LIN {X 0,Y 308.956,Z 964.973,A -85,B 0,C 180,E1 8655.681,E2 8655.681} C_VEL
LIN {X 0,Y 317.199,Z 943.348,A -85,B 0,C 180,E1 8654.6,E2 8654.6} C_VEL
LIN {X 0,Y 323.578,Z 923.233,A -85,B 0,C 180,E1 8653.806,E2 8653.806} C_VEL
LIN {X 0,Y 329.227,Z 900.533,A -85,B 0,C 180,E1 8653.113,E2 8653.113} C_VEL
LIN {X 0,Y 333.474,Z 877.732,A -85,B 0,C 180,E1 8652.592,E2 8652.592} C_VEL
LIN {X 0,Y 338.815,Z 829.601,A -85,B 0,C 180,E1 8651.724,E2 8651.724} C_VEL
LIN {X 0,Y 347.713,Z 744.532,A -85,B 0,C 180,E1 8650.195,E2 8650.195} C_VEL
LIN {X 0,Y 346.209,Z 741.442,A -85,B 0,C 180,E1 8648.219,E2 8648.219} C_VEL
LIN {X 0,Y 345.828,Z 740.56,A -85,B 0,C 180,E1 8647.617,E2 8647.617} C_VEL
LIN {X 0,Y 345.026,Z 739.757,A -85,B 0,C 180,E1 8646.353,E2 8646.353} C_VEL
LIN {X 0,Y 343.82,Z 741.091,A -85,B 0,C 180,E1 8644.432,E2 8644.432} C_VEL
LIN {X 0,Y 342.845,Z 743.031,A -85,B 0,C 180,E1 8642.109,E2 8642.109} C_VEL
LIN {X 0,Y 342.775,Z 743.064,A -85,B 0,C 180,E1 8641.733,E2 8641.733} C_VEL
LIN {X 0,Y 342.85,Z 743.346,A -85,B 0,C 180,E1 8638.162,E2 8638.162} C_VEL
LIN {X 0,Y 344.465,Z 747.751,A -85,B 0,C 180,E1 8633.5,E2 8633.5} C_VEL
LIN {X 0,Y 345.843,Z 750.98,A -85,B 0,C 180,E1 8631.351,E2 8631.351} C_VEL
LIN {X 0,Y 331.864,Z 879.656,A -85,B 0,C 180,E1 8629.105,E2 8629.105} C_VEL
LIN {X 0,Y 327.557,Z 903.577,A -85,B 0,C 180,E1 8628.614,E2 8628.614} C_VEL
LIN {X 0,Y 321.932,Z 926.311,A -85,B 0,C 180,E1 8628.05,E2 8628.05} C_VEL
LIN {X 0,Y 315.075,Z 947.567,A -85,B 0,C 180,E1 8627.352,E2 8627.352} C_VEL
LIN {X 0,Y 306.548,Z 969.68,A -85,B 0,C 180,E1 8626.404,E2 8626.404} C_VEL
LIN {X 0,Y 297.655,Z 989.023,A -85,B 0,C 180,E1 8625.336,E2 8625.336} C_VEL
LIN {X 0,Y 286.855,Z 1009.539,A -85,B 0,C 180,E1 8623.906,E2 8623.906} C_VEL
LIN {X 0,Y 275.629,Z 1028.122,A -85,B 0,C 180,E1 8622.26,E2 8622.26} C_VEL
LIN {X 0,Y 262.429,Z 1047.52,A -85,B 0,C 180,E1 8620.071,E2 8620.071} C_VEL
LIN {X 0,Y 249.67,Z 1064.385,A -85,B 0,C 180,E1 8617.639,E2 8617.639} C_VEL
LIN {X 0,Y 236.423,Z 1080.167,A -85,B 0,C 180,E1 8614.715,E2 8614.715} C_VEL
LIN {X 0,Y 223.404,Z 1094.596,A -85,B 0,C 180,E1 8611.307,E2 8611.307} C_VEL
LIN {X 0,Y 210.28,Z 1107.943,A -85,B 0,C 180,E1 8607.177,E2 8607.177} C_VEL
LIN {X 0,Y 197.502,Z 1120.368,A -85,B 0,C 180,E1 8602.162,E2 8602.162} C_VEL
LIN {X 0,Y 186.671,Z 1130.485,A -85,B 0,C 180,E1 8596.718,E2 8596.718} C_VEL
LIN {X 0,Y 176.025,Z 1140.477,A -85,B 0,C 180,E1 8589.507,E2 8589.507} C_VEL
LIN {X 0,Y 168.922,Z 1147.539,A -85,B 0,C 180,E1 8582.59,E2 8582.59} C_VEL
LIN {X 0,Y 163.641,Z 1153.455,A -85,B 0,C 180,E1 8574.549,E2 8574.549} C_VEL
LIN {X 0,Y 161.075,Z 1157.231,A -85,B 0,C 180,E1 8567.334,E2 8567.334} C_VEL
LIN {X 0,Y 160.092,Z 1159.786,A -85,B 0,C 180,E1 8559.707,E2 8559.707} C_VEL
LIN {X 0,Y 160.029,Z 1160.788,A -85,B 0,C 180,E1 8553.581,E2 8553.581} C_VEL
LIN {X 0,Y 160.056,Z 1160.906,A -85,B 0,C 180,E1 8548.17,E2 8548.17} C_VEL
LIN {X 0,Y 160.02,Z 1160.217,A -85,B 0,C 180,E1 8542.459,E2 8542.459} C_VEL
LIN {X 0,Y 160.43,Z 1158.581,A -85,B 0,C 180,E1 8536.3,E2 8536.3} C_VEL
LIN {X 0,Y 162.397,Z 1155.157,A -85,B 0,C 180,E1 8528.32,E2 8528.32} C_VEL
LIN {X 0,Y 166.539,Z 1150.008,A -85,B 0,C 180,E1 8520.507,E2 8520.507} C_VEL
LIN {X 0,Y 173.063,Z 1143.346,A -85,B 0,C 180,E1 8513.068,E2 8513.068} C_VEL
LIN {X 0,Y 181.484,Z 1135.255,A -85,B 0,C 180,E1 8506.474,E2 8506.474} C_VEL
LIN {X 0,Y 192.44,Z 1125.043,A -85,B 0,C 180,E1 8500.201,E2 8500.201} C_VEL
LIN {X 0,Y 204.092,Z 1113.937,A -85,B 0,C 180,E1 8495.099,E2 8495.099} C_VEL
LIN {X 0,Y 217.805,Z 1100.223,A -85,B 0,C 180,E1 8490.339,E2 8490.339} C_VEL
LIN {X 0,Y 231.353,Z 1085.847,A -85,B 0,C 180,E1 8486.539,E2 8486.539} C_VEL
LIN {X 0,Y 245.008,Z 1069.898,A -85,B 0,C 180,E1 8483.332,E2 8483.332} C_VEL
LIN {X 0,Y 258.548,Z 1052.656,A -85,B 0,C 180,E1 8480.63,E2 8480.63} C_VEL
LIN {X 0,Y 270.101,Z 1036.297,A -85,B 0,C 180,E1 8478.617,E2 8478.617} C_VEL
LIN {X 0,Y 282.833,Z 1016.155,A -85,B 0,C 180,E1 8476.657,E2 8476.657} C_VEL
LIN {X 0,Y 292.819,Z 998.254,A -85,B 0,C 180,E1 8475.283,E2 8475.283} C_VEL
LIN {X 0,Y 302.973,Z 977.385,A -85,B 0,C 180,E1 8474.009,E2 8474.009} C_VEL
LIN {X 0,Y 311.029,Z 958.092,A -85,B 0,C 180,E1 8473.078,E2 8473.078} C_VEL
LIN {X 0,Y 319.051,Z 935.046,A -85,B 0,C 180,E1 8472.219,E2 8472.219} C_VEL
LIN {X 0,Y 325.38,Z 912.51,A -85,B 0,C 180,E1 8471.595,E2 8471.595} C_VEL
LIN {X 0,Y 330.153,Z 889.153,A -85,B 0,C 180,E1 8471.088,E2 8471.088} C_VEL
LIN {X 0,Y 333.618,Z 863.695,A -85,B 0,C 180,E1 8470.613,E2 8470.613} C_VEL
LIN {X 0,Y 345.663,Z 750.594,A -85,B 0,C 180,E1 8468.63,E2 8468.63} C_VEL
LIN {X 0,Y 343.916,Z 746.807,A -85,B 0,C 180,E1 8465.84,E2 8465.84} C_VEL
LIN {X 0,Y 342.587,Z 742.997,A -85,B 0,C 180,E1 8461.505,E2 8461.505} C_VEL
LIN {X 0,Y 342.658,Z 743.159,A -85,B 0,C 180,E1 8457.491,E2 8457.491} C_VEL
LIN {X 0,Y 344.322,Z 747.735,A -85,B 0,C 180,E1 8452.827,E2 8452.827} C_VEL
LIN {X 0,Y 345.579,Z 750.709,A -85,B 0,C 180,E1 8450.872,E2 8450.872} C_VEL
LIN {X 0,Y 332.039,Z 874.961,A -85,B 0,C 180,E1 8448.717,E2 8448.717} C_VEL
LIN {X 0,Y 327.811,Z 898.507,A -85,B 0,C 180,E1 8448.211,E2 8448.211} C_VEL
LIN {X 0,Y 322.548,Z 920.18,A -85,B 0,C 180,E1 8447.599,E2 8447.599} C_VEL
LIN {X 0,Y 315.6,Z 942.141,A -85,B 0,C 180,E1 8446.78,E2 8446.78} C_VEL
LIN {X 0,Y 307.409,Z 963.644,A -85,B 0,C 180,E1 8445.759,E2 8445.759} C_VEL
LIN {X 0,Y 298.233,Z 983.67,A -85,B 0,C 180,E1 8444.555,E2 8444.555} C_VEL
LIN {X 0,Y 287.107,Z 1004.651,A -85,B 0,C 180,E1 8442.968,E2 8442.968} C_VEL
LIN {X 0,Y 276.119,Z 1022.72,A -85,B 0,C 180,E1 8441.251,E2 8441.251} C_VEL
LIN {X 0,Y 263.396,Z 1041.188,A -85,B 0,C 180,E1 8439.041,E2 8439.041} C_VEL
LIN {X 0,Y 250.7,Z 1057.772,A -85,B 0,C 180,E1 8436.537,E2 8436.537} C_VEL
LIN {X 0,Y 237.755,Z 1072.886,A -85,B 0,C 180,E1 8433.607,E2 8433.607} C_VEL
LIN {X 0,Y 224.49,Z 1087.223,A -85,B 0,C 180,E1 8430.076,E2 8430.076} C_VEL
LIN {X 0,Y 211.99,Z 1099.548,A -85,B 0,C 180,E1 8426.112,E2 8426.112} C_VEL
LIN {X 0,Y 199.154,Z 1111.528,A -85,B 0,C 180,E1 8421.096,E2 8421.096} C_VEL
LIN {X 0,Y 188.389,Z 1121.067,A -85,B 0,C 180,E1 8415.768,E2 8415.768} C_VEL
LIN {X 0,Y 178.024,Z 1130.106,A -85,B 0,C 180,E1 8408.98,E2 8408.98} C_VEL
LIN {X 0,Y 170.33,Z 1137.007,A -85,B 0,C 180,E1 8401.893,E2 8401.893} C_VEL
LIN {X 0,Y 164.905,Z 1142.188,A -85,B 0,C 180,E1 8394.35,E2 8394.35} C_VEL
LIN {X 0,Y 161.901,Z 1145.626,A -85,B 0,C 180,E1 8387.245,E2 8387.245} C_VEL
LIN {X 0,Y 160.409,Z 1147.984,A -85,B 0,C 180,E1 8379.328,E2 8379.328} C_VEL
LIN {X 0,Y 160.08,Z 1148.822,A -85,B 0,C 180,E1 8373.223,E2 8373.223} C_VEL
LIN {X 0,Y 160.075,Z 1148.894,A -85,B 0,C 180,E1 8367.853,E2 8367.853} C_VEL
LIN {X 0,Y 160.266,Z 1148.264,A -85,B 0,C 180,E1 8362.112,E2 8362.112} C_VEL
LIN {X 0,Y 161.155,Z 1146.683,A -85,B 0,C 180,E1 8355.631,E2 8355.631} C_VEL
LIN {X 0,Y 163.961,Z 1143.253,A -85,B 0,C 180,E1 8347.408,E2 8347.408} C_VEL
LIN {X 0,Y 168.558,Z 1138.646,A -85,B 0,C 180,E1 8340.115,E2 8340.115} C_VEL
LIN {X 0,Y 176.373,Z 1131.605,A -85,B 0,C 180,E1 8332.248,E2 8332.248} C_VEL
LIN {X 0,Y 185.632,Z 1123.595,A -85,B 0,C 180,E1 8325.756,E2 8325.756} C_VEL
LIN {X 0,Y 196.778,Z 1113.715,A -85,B 0,C 180,E1 8319.893,E2 8319.893} C_VEL
LIN {X 0,Y 208.697,Z 1102.877,A -85,B 0,C 180,E1 8314.99,E2 8314.99} C_VEL
LIN {X 0,Y 221.196,Z 1090.62,A -85,B 0,C 180,E1 8310.813,E2 8310.813} C_VEL
LIN {X 0,Y 234.698,Z 1076.5,A -85,B 0,C 180,E1 8307.079,E2 8307.079} C_VEL
LIN {X 0,Y 247.489,Z 1061.776,A -85,B 0,C 180,E1 8304.071,E2 8304.071} C_VEL
LIN {X 0,Y 261.675,Z 1043.747,A -85,B 0,C 180,E1 8301.201,E2 8301.201} C_VEL
LIN {X 0,Y 273.94,Z 1026.37,A -85,B 0,C 180,E1 8299.033,E2 8299.033} C_VEL
LIN {X 0,Y 285.687,Z 1007.387,A -85,B 0,C 180,E1 8297.166,E2 8297.166} C_VEL
LIN {X 0,Y 296.411,Z 987.815,A -85,B 0,C 180,E1 8295.624,E2 8295.624} C_VEL
LIN {X 0,Y 305.56,Z 968.258,A -85,B 0,C 180,E1 8294.4,E2 8294.4} C_VEL
LIN {X 0,Y 313.944,Z 947.472,A -85,B 0,C 180,E1 8293.354,E2 8293.354} C_VEL
LIN {X 0,Y 320.615,Z 927.28,A -85,B 0,C 180,E1 8292.55,E2 8292.55} C_VEL
LIN {X 0,Y 326.683,Z 904.611,A -85,B 0,C 180,E1 8291.843,E2 8291.843} C_VEL
LIN {X 0,Y 331.028,Z 882.586,A -85,B 0,C 180,E1 8291.335,E2 8291.335} C_VEL
LIN {X 0,Y 334.95,Z 851.804,A -85,B 0,C 180,E1 8290.773,E2 8290.773} C_VEL
LIN {X 0,Y 345.775,Z 750.614,A -85,B 0,C 180,E1 8289.012,E2 8289.012} C_VEL
LIN {X 0,Y 344.121,Z 747.017,A -85,B 0,C 180,E1 8286.339,E2 8286.339} C_VEL
LIN {X 0,Y 342.791,Z 743.072,A -85,B 0,C 180,E1 8281.839,E2 8281.839} C_VEL
LIN {X 0,Y 342.775,Z 743.064,A -85,B 0,C 180,E1 8281.733,E2 8281.733} C_VEL
LIN {X 0,Y 342.552,Z 743.97,A -85,B 0,C 180,E1 8280.536,E2 8280.536} C_VEL
LIN {X 0,Y 342.205,Z 747.569,A -85,B 0,C 180,E1 8278.86,E2 8278.86} C_VEL
LIN {X 0,Y 342.137,Z 752.531,A -85,B 0,C 180,E1 8276.736,E2 8276.736} C_VEL
LIN {X 0,Y 342.317,Z 753.491,A -85,B 0,C 180,E1 8275.998,E2 8275.998} C_VEL
LIN {X 0,Y 343.338,Z 755.566,A -85,B 0,C 180,E1 8273.731,E2 8273.731} C_VEL
LIN {X 0,Y 343.982,Z 757.422,A -85,B 0,C 180,E1 8272.561,E2 8272.561} C_VEL
LIN {X 0,Y 330.418,Z 879.53,A -85,B 0,C 180,E1 8270.472,E2 8270.472} C_VEL
LIN {X 0,Y 326.064,Z 903.288,A -85,B 0,C 180,E1 8270,E2 8270} C_VEL
LIN {X 0,Y 320.36,Z 926.018,A -85,B 0,C 180,E1 8269.461,E2 8269.461} C_VEL
LIN {X 0,Y 313.382,Z 947.333,A -85,B 0,C 180,E1 8268.793,E2 8268.793} C_VEL
LIN {X 0,Y 304.611,Z 969.672,A -85,B 0,C 180,E1 8267.874,E2 8267.874} C_VEL
LIN {X 0,Y 295.249,Z 989.63,A -85,B 0,C 180,E1 8266.809,E2 8266.809} C_VEL
LIN {X 0,Y 283.677,Z 1010.946,A -85,B 0,C 180,E1 8265.355,E2 8265.355} C_VEL
LIN {X 0,Y 272.365,Z 1029.178,A -85,B 0,C 180,E1 8263.771,E2 8263.771} C_VEL
LIN {X 0,Y 259.1,Z 1048.055,A -85,B 0,C 180,E1 8261.677,E2 8261.677} C_VEL
LIN {X 0,Y 245.881,Z 1065.031,A -85,B 0,C 180,E1 8259.273,E2 8259.273} C_VEL
LIN {X 0,Y 232.252,Z 1080.669,A -85,B 0,C 180,E1 8256.399,E2 8256.399} C_VEL
LIN {X 0,Y 218.047,Z 1095.745,A -85,B 0,C 180,E1 8252.821,E2 8252.821} C_VEL
LIN {X 0,Y 204.685,Z 1108.754,A -85,B 0,C 180,E1 8248.743,E2 8248.743} C_VEL
LIN {X 0,Y 190.654,Z 1121.637,A -85,B 0,C 180,E1 8243.358,E2 8243.358} C_VEL
LIN {X 0,Y 178.852,Z 1132.136,A -85,B 0,C 180,E1 8237.435,E2 8237.435} C_VEL
LIN {X 0,Y 168.815,Z 1140.894,A -85,B 0,C 180,E1 8230.655,E2 8230.655} C_VEL
LIN {X 0,Y 160.948,Z 1148.225,A -85,B 0,C 180,E1 8223.003,E2 8223.003} C_VEL
LIN {X 0,Y 155.771,Z 1153.578,A -85,B 0,C 180,E1 8215.064,E2 8215.064} C_VEL
LIN {X 0,Y 152.916,Z 1157.562,A -85,B 0,C 180,E1 8206.719,E2 8206.719} C_VEL
LIN {X 0,Y 152.077,Z 1159.704,A -85,B 0,C 180,E1 8199.078,E2 8199.078} C_VEL
LIN {X 0,Y 152.038,Z 1160.538,A -85,B 0,C 180,E1 8193.015,E2 8193.015} C_VEL
LIN {X 0,Y 152.051,Z 1160.584,A -85,B 0,C 180,E1 8187.738,E2 8187.738} C_VEL
LIN {X 0,Y 152.053,Z 1159.842,A -85,B 0,C 180,E1 8181.681,E2 8181.681} C_VEL
LIN {X 0,Y 152.633,Z 1158.032,A -85,B 0,C 180,E1 8174.809,E2 8174.809} C_VEL
LIN {X 0,Y 155.243,Z 1154.199,A -85,B 0,C 180,E1 8166.06,E2 8166.06} C_VEL
LIN {X 0,Y 159.891,Z 1149.165,A -85,B 0,C 180,E1 8158.312,E2 8158.312} C_VEL
LIN {X 0,Y 168.005,Z 1141.571,A -85,B 0,C 180,E1 8150.002,E2 8150.002} C_VEL
LIN {X 0,Y 177.961,Z 1132.853,A -85,B 0,C 180,E1 8143.079,E2 8143.079} C_VEL
LIN {X 0,Y 189.466,Z 1122.616,A -85,B 0,C 180,E1 8137.167,E2 8137.167} C_VEL
LIN {X 0,Y 202.007,Z 1111.246,A -85,B 0,C 180,E1 8132.178,E2 8132.178} C_VEL
LIN {X 0,Y 215.138,Z 1098.48,A -85,B 0,C 180,E1 8127.988,E2 8127.988} C_VEL
LIN {X 0,Y 229.277,Z 1083.832,A -85,B 0,C 180,E1 8124.294,E2 8124.294} C_VEL
LIN {X 0,Y 242.238,Z 1069.114,A -85,B 0,C 180,E1 8121.442,E2 8121.442} C_VEL
LIN {X 0,Y 256.582,Z 1051.219,A -85,B 0,C 180,E1 8118.747,E2 8118.747} C_VEL
LIN {X 0,Y 268.841,Z 1034.181,A -85,B 0,C 180,E1 8116.75,E2 8116.75} C_VEL
LIN {X 0,Y 281.469,Z 1014.36,A -85,B 0,C 180,E1 8114.931,E2 8114.931} C_VEL
LIN {X 0,Y 292.561,Z 994.673,A -85,B 0,C 180,E1 8113.512,E2 8113.512} C_VEL
LIN {X 0,Y 302.467,Z 974.041,A -85,B 0,C 180,E1 8112.354,E2 8112.354} C_VEL
LIN {X 0,Y 311.134,Z 953.139,A -85,B 0,C 180,E1 8111.432,E2 8111.432} C_VEL
LIN {X 0,Y 318.265,Z 932.103,A -85,B 0,C 180,E1 8110.72,E2 8110.72} C_VEL
LIN {X 0,Y 324.621,Z 908.927,A -85,B 0,C 180,E1 8110.128,E2 8110.128} C_VEL
LIN {X 0,Y 329.1,Z 886.554,A -85,B 0,C 180,E1 8109.667,E2 8109.667} C_VEL
LIN {X 0,Y 333.092,Z 855.375,A -85,B 0,C 180,E1 8109.111,E2 8109.111} C_VEL
LIN {X 0,Y 343.806,Z 757.094,A -85,B 0,C 180,E1 8107.435,E2 8107.435} C_VEL
LIN {X 0,Y 342.761,Z 754.556,A -85,B 0,C 180,E1 8105.524,E2 8105.524} C_VEL
LIN {X 0,Y 341.613,Z 750.938,A -85,B 0,C 180,E1 8101.509,E2 8101.509} C_VEL
LIN {X 0,Y 341.652,Z 751.052,A -85,B 0,C 180,E1 8097.651,E2 8097.651} C_VEL
LIN {X 0,Y 343.193,Z 755.551,A -85,B 0,C 180,E1 8093.055,E2 8093.055} C_VEL
LIN {X 0,Y 343.719,Z 757.217,A -85,B 0,C 180,E1 8092.081,E2 8092.081} C_VEL
LIN {X 0,Y 330.545,Z 875.455,A -85,B 0,C 180,E1 8090.073,E2 8090.073} C_VEL
LIN {X 0,Y 326.269,Z 898.825,A -85,B 0,C 180,E1 8089.587,E2 8089.587} C_VEL
LIN {X 0,Y 320.865,Z 920.708,A -85,B 0,C 180,E1 8088.991,E2 8088.991} C_VEL
LIN {X 0,Y 313.907,Z 942.315,A -85,B 0,C 180,E1 8088.214,E2 8088.214} C_VEL
LIN {X 0,Y 305.528,Z 963.953,A -85,B 0,C 180,E1 8087.223,E2 8087.223} C_VEL
LIN {X 0,Y 296.185,Z 983.979,A -85,B 0,C 180,E1 8086.061,E2 8086.061} C_VEL
LIN {X 0,Y 284.844,Z 1004.952,A -85,B 0,C 180,E1 8084.527,E2 8084.527} C_VEL
LIN {X 0,Y 273.641,Z 1022.989,A -85,B 0,C 180,E1 8082.867,E2 8082.867} C_VEL
LIN {X 0,Y 260.589,Z 1041.497,A -85,B 0,C 180,E1 8080.717,E2 8080.717} C_VEL
LIN {X 0,Y 247.554,Z 1058.082,A -85,B 0,C 180,E1 8078.275,E2 8078.275} C_VEL
LIN {X 0,Y 234.218,Z 1073.197,A -85,B 0,C 180,E1 8075.408,E2 8075.408} C_VEL
LIN {X 0,Y 220.792,Z 1087.25,A -85,B 0,C 180,E1 8072.016,E2 8072.016} C_VEL
LIN {X 0,Y 207.408,Z 1099.944,A -85,B 0,C 180,E1 8067.975,E2 8067.975} C_VEL
LIN {X 0,Y 194.063,Z 1111.84,A -85,B 0,C 180,E1 8062.998,E2 8062.998} C_VEL
LIN {X 0,Y 182.713,Z 1121.378,A -85,B 0,C 180,E1 8057.627,E2 8057.627} C_VEL
LIN {X 0,Y 171.675,Z 1130.417,A -85,B 0,C 180,E1 8050.717,E2 8050.717} C_VEL
LIN {X 0,Y 163.391,Z 1137.317,A -85,B 0,C 180,E1 8043.42,E2 8043.42} C_VEL
LIN {X 0,Y 157.473,Z 1142.496,A -85,B 0,C 180,E1 8035.58,E2 8035.58} C_VEL
LIN {X 0,Y 154.146,Z 1145.932,A -85,B 0,C 180,E1 8028.141,E2 8028.141} C_VEL
LIN {X 0,Y 152.469,Z 1148.286,A -85,B 0,C 180,E1 8019.818,E2 8019.818} C_VEL
LIN {X 0,Y 152.088,Z 1149.122,A -85,B 0,C 180,E1 8013.393,E2 8013.393} C_VEL
LIN {X 0,Y 152.08,Z 1149.193,A -85,B 0,C 180,E1 8007.74,E2 8007.74} C_VEL
LIN {X 0,Y 152.298,Z 1148.566,A -85,B 0,C 180,E1 8001.696,E2 8001.696} C_VEL
LIN {X 0,Y 153.314,Z 1146.977,A -85,B 0,C 180,E1 7994.843,E2 7994.843} C_VEL
LIN {X 0,Y 156.598,Z 1143.386,A -85,B 0,C 180,E1 7985.93,E2 7985.93} C_VEL
LIN {X 0,Y 161.764,Z 1138.71,A -85,B 0,C 180,E1 7978.307,E2 7978.307} C_VEL
LIN {X 0,Y 170.206,Z 1131.672,A -85,B 0,C 180,E1 7970.314,E2 7970.314} C_VEL
LIN {X 0,Y 180.54,Z 1123.32,A -85,B 0,C 180,E1 7963.49,E2 7963.49} C_VEL
LIN {X 0,Y 192.161,Z 1113.521,A -85,B 0,C 180,E1 7957.732,E2 7957.732} C_VEL
LIN {X 0,Y 205.389,Z 1101.942,A -85,B 0,C 180,E1 7952.629,E2 7952.629} C_VEL
LIN {X 0,Y 218.517,Z 1089.551,A -85,B 0,C 180,E1 7948.535,E2 7948.535} C_VEL
LIN {X 0,Y 232.582,Z 1075.142,A -85,B 0,C 180,E1 7944.896,E2 7944.896} C_VEL
LIN {X 0,Y 245.848,Z 1060.255,A -85,B 0,C 180,E1 7941.987,E2 7941.987} C_VEL
LIN {X 0,Y 259.246,Z 1043.501,A -85,B 0,C 180,E1 7939.441,E2 7939.441} C_VEL
LIN {X 0,Y 271.901,Z 1025.952,A -85,B 0,C 180,E1 7937.33,E2 7937.33} C_VEL
LIN {X 0,Y 283.926,Z 1006.803,A -85,B 0,C 180,E1 7935.524,E2 7935.524} C_VEL
LIN {X 0,Y 295.215,Z 986.325,A -85,B 0,C 180,E1 7933.99,E2 7933.99} C_VEL
LIN {X 0,Y 304.546,Z 966.563,A -85,B 0,C 180,E1 7932.817,E2 7932.817} C_VEL
LIN {X 0,Y 313.531,Z 943.934,A -85,B 0,C 180,E1 7931.754,E2 7931.754} C_VEL
LIN {X 0,Y 320.129,Z 923.816,A -85,B 0,C 180,E1 7931.016,E2 7931.016} C_VEL
LIN {X 0,Y 325.967,Z 901.107,A -85,B 0,C 180,E1 7930.371,E2 7930.371} C_VEL
LIN {X 0,Y 330.355,Z 878.298,A -85,B 0,C 180,E1 7929.882,E2 7929.882} C_VEL
LIN {X 0,Y 335.986,Z 829.62,A -85,B 0,C 180,E1 7929.041,E2 7929.041} C_VEL
LIN {X 0,Y 343.932,Z 757.115,A -85,B 0,C 180,E1 7927.812,E2 7927.812} C_VEL
LIN {X 0,Y 342.968,Z 754.768,A -85,B 0,C 180,E1 7926.025,E2 7926.025} C_VEL
LIN {X 0,Y 341.792,Z 751,A -85,B 0,C 180,E1 7921.677,E2 7921.677} C_VEL
LIN {X 0,Y 341.847,Z 751.235,A -85,B 0,C 180,E1 7918.324,E2 7918.324} C_VEL
LIN {X 0,Y 342.317,Z 753.491,A -85,B 0,C 180,E1 7915.998,E2 7915.998} C_VEL
LIN {X 0,Y 342.457,Z 755.145,A -85,B 0,C 180,E1 7915.284,E2 7915.284} C_VEL
LIN {X 0,Y 342.387,Z 758.764,A -85,B 0,C 180,E1 7914.605,E2 7914.605} C_VEL
LIN {X 0,Y 342.063,Z 764.238,A -85,B 0,C 180,E1 7914.036,E2 7914.036} C_VEL
LIN {X 0,Y 341.441,Z 771.258,A -85,B 0,C 180,E1 7913.669,E2 7913.669} C_VEL
LIN {X 0,Y 341.266,Z 772.878,A -85,B 0,C 180,E1 7913.632,E2 7913.632} C_VEL
LIN {X 0,Y 329.153,Z 879.464,A -85,B 0,C 180,E1 7911.85,E2 7911.85} C_VEL
LIN {X 0,Y 324.734,Z 903.13,A -85,B 0,C 180,E1 7911.396,E2 7911.396} C_VEL
LIN {X 0,Y 318.984,Z 925.725,A -85,B 0,C 180,E1 7910.884,E2 7910.884} C_VEL
LIN {X 0,Y 311.957,Z 946.909,A -85,B 0,C 180,E1 7910.255,E2 7910.255} C_VEL
LIN {X 0,Y 303.142,Z 969.084,A -85,B 0,C 180,E1 7909.388,E2 7909.388} C_VEL
LIN {X 0,Y 293.498,Z 989.33,A -85,B 0,C 180,E1 7908.357,E2 7908.357} C_VEL
LIN {X 0,Y 281.85,Z 1010.429,A -85,B 0,C 180,E1 7906.981,E2 7906.981} C_VEL
LIN {X 0,Y 270.582,Z 1028.268,A -85,B 0,C 180,E1 7905.499,E2 7905.499} C_VEL
LIN {X 0,Y 257.172,Z 1047.039,A -85,B 0,C 180,E1 7903.512,E2 7903.512} C_VEL
LIN {X 0,Y 243.904,Z 1063.698,A -85,B 0,C 180,E1 7901.254,E2 7901.254} C_VEL
LIN {X 0,Y 229.961,Z 1079.378,A -85,B 0,C 180,E1 7898.506,E2 7898.506} C_VEL
LIN {X 0,Y 215.874,Z 1093.974,A -85,B 0,C 180,E1 7895.204,E2 7895.204} C_VEL
LIN {X 0,Y 201.879,Z 1107.147,A -85,B 0,C 180,E1 7891.239,E2 7891.239} C_VEL
LIN {X 0,Y 188.32,Z 1119.215,A -85,B 0,C 180,E1 7886.466,E2 7886.466} C_VEL
LIN {X 0,Y 175.629,Z 1129.818,A -85,B 0,C 180,E1 7880.736,E2 7880.736} C_VEL
LIN {X 0,Y 163.535,Z 1139.774,A -85,B 0,C 180,E1 7873.318,E2 7873.318} C_VEL
LIN {X 0,Y 155.106,Z 1146.915,A -85,B 0,C 180,E1 7865.916,E2 7865.916} C_VEL
LIN {X 0,Y 148.735,Z 1152.835,A -85,B 0,C 180,E1 7857.201,E2 7857.201} C_VEL
LIN {X 0,Y 145.388,Z 1156.785,A -85,B 0,C 180,E1 7848.857,E2 7848.857} C_VEL
LIN {X 0,Y 144.12,Z 1159.253,A -85,B 0,C 180,E1 7840.391,E2 7840.391} C_VEL
LIN {X 0,Y 144.037,Z 1160.187,A -85,B 0,C 180,E1 7833.98,E2 7833.98} C_VEL
LIN {X 0,Y 144.068,Z 1160.332,A -85,B 0,C 180,E1 7828.408,E2 7828.408} C_VEL
LIN {X 0,Y 144.039,Z 1159.685,A -85,B 0,C 180,E1 7822.019,E2 7822.019} C_VEL
LIN {X 0,Y 144.563,Z 1158.09,A -85,B 0,C 180,E1 7815.172,E2 7815.172} C_VEL
LIN {X 0,Y 146.846,Z 1154.905,A -85,B 0,C 180,E1 7806.738,E2 7806.738} C_VEL
LIN {X 0,Y 151.697,Z 1149.913,A -85,B 0,C 180,E1 7798.176,E2 7798.176} C_VEL
LIN {X 0,Y 159.505,Z 1143.153,A -85,B 0,C 180,E1 7789.884,E2 7789.884} C_VEL
LIN {X 0,Y 169.71,Z 1134.623,A -85,B 0,C 180,E1 7782.569,E2 7782.569} C_VEL
LIN {X 0,Y 182.061,Z 1124.41,A -85,B 0,C 180,E1 7776.164,E2 7776.164} C_VEL
LIN {X 0,Y 194.926,Z 1113.304,A -85,B 0,C 180,E1 7771.059,E2 7771.059} C_VEL
LIN {X 0,Y 209.856,Z 1099.592,A -85,B 0,C 180,E1 7766.396,E2 7766.396} C_VEL
LIN {X 0,Y 224.4,Z 1085.217,A -85,B 0,C 180,E1 7762.728,E2 7762.728} C_VEL
LIN {X 0,Y 238.914,Z 1069.269,A -85,B 0,C 180,E1 7759.67,E2 7759.67} C_VEL
LIN {X 0,Y 253.193,Z 1052.029,A -85,B 0,C 180,E1 7757.123,E2 7757.123} C_VEL
LIN {X 0,Y 265.738,Z 1035.057,A -85,B 0,C 180,E1 7755.179,E2 7755.179} C_VEL
LIN {X 0,Y 278.997,Z 1014.833,A -85,B 0,C 180,E1 7753.369,E2 7753.369} C_VEL
LIN {X 0,Y 289.807,Z 996.081,A -85,B 0,C 180,E1 7752.058,E2 7752.058} C_VEL
LIN {X 0,Y 299.913,Z 975.753,A -85,B 0,C 180,E1 7750.941,E2 7750.941} C_VEL
LIN {X 0,Y 308.236,Z 956.333,A -85,B 0,C 180,E1 7750.098,E2 7750.098} C_VEL
LIN {X 0,Y 316.159,Z 934.019,A -85,B 0,C 180,E1 7749.349,E2 7749.349} C_VEL
LIN {X 0,Y 322.678,Z 911.336,A -85,B 0,C 180,E1 7748.781,E2 7748.781} C_VEL
LIN {X 0,Y 327.525,Z 888.028,A -85,B 0,C 180,E1 7748.314,E2 7748.314} C_VEL
LIN {X 0,Y 331.228,Z 861.254,A -85,B 0,C 180,E1 7747.843,E2 7747.843} C_VEL
LIN {X 0,Y 342.102,Z 763.458,A -85,B 0,C 180,E1 7746.208,E2 7746.208} C_VEL
LIN {X 0,Y 341.393,Z 761.898,A -85,B 0,C 180,E1 7744.703,E2 7744.703} C_VEL
LIN {X 0,Y 340.609,Z 758.867,A -85,B 0,C 180,E1 7741.345,E2 7741.345} C_VEL
LIN {X 0,Y 340.661,Z 759.127,A -85,B 0,C 180,E1 7737.645,E2 7737.645} C_VEL
LIN {X 0,Y 342.056,Z 763.336,A -85,B 0,C 180,E1 7733.311,E2 7733.311} C_VEL
LIN {X 0,Y 329.26,Z 875.777,A -85,B 0,C 180,E1 7731.445,E2 7731.445} C_VEL
LIN {X 0,Y 324.911,Z 899.169,A -85,B 0,C 180,E1 7730.975,E2 7730.975} C_VEL
LIN {X 0,Y 319.43,Z 921.02,A -85,B 0,C 180,E1 7730.403,E2 7730.403} C_VEL
LIN {X 0,Y 312.322,Z 942.743,A -85,B 0,C 180,E1 7729.652,E2 7729.652} C_VEL
LIN {X 0,Y 303.848,Z 964.261,A -85,B 0,C 180,E1 7728.704,E2 7728.704} C_VEL
LIN {X 0,Y 294.345,Z 984.287,A -85,B 0,C 180,E1 7727.586,E2 7727.586} C_VEL
LIN {X 0,Y 283.186,Z 1004.613,A -85,B 0,C 180,E1 7726.161,E2 7726.161} C_VEL
LIN {X 0,Y 271.767,Z 1022.677,A -85,B 0,C 180,E1 7724.566,E2 7724.566} C_VEL
LIN {X 0,Y 258.437,Z 1041.258,A -85,B 0,C 180,E1 7722.495,E2 7722.495} C_VEL
LIN {X 0,Y 245.465,Z 1057.392,A -85,B 0,C 180,E1 7720.212,E2 7720.212} C_VEL
LIN {X 0,Y 231.541,Z 1072.855,A -85,B 0,C 180,E1 7717.397,E2 7717.397} C_VEL
LIN {X 0,Y 217.797,Z 1086.825,A -85,B 0,C 180,E1 7714.133,E2 7714.133} C_VEL
LIN {X 0,Y 203.943,Z 1099.55,A -85,B 0,C 180,E1 7710.202,E2 7710.202} C_VEL
LIN {X 0,Y 190.29,Z 1111.297,A -85,B 0,C 180,E1 7705.425,E2 7705.425} C_VEL
LIN {X 0,Y 177.802,Z 1121.243,A -85,B 0,C 180,E1 7699.89,E2 7699.89} C_VEL
LIN {X 0,Y 165.954,Z 1130.387,A -85,B 0,C 180,E1 7692.909,E2 7692.909} C_VEL
LIN {X 0,Y 157.282,Z 1137.042,A -85,B 0,C 180,E1 7685.794,E2 7685.794} C_VEL
LIN {X 0,Y 150.357,Z 1142.607,A -85,B 0,C 180,E1 7677.314,E2 7677.314} C_VEL
LIN {X 0,Y 146.565,Z 1146.086,A -85,B 0,C 180,E1 7669.53,E2 7669.53} C_VEL
LIN {X 0,Y 144.577,Z 1148.526,A -85,B 0,C 180,E1 7660.763,E2 7660.763} C_VEL
LIN {X 0,Y 144.097,Z 1149.423,A -85,B 0,C 180,E1 7653.581,E2 7653.581} C_VEL
LIN {X 0,Y 144.085,Z 1149.494,A -85,B 0,C 180,E1 7647.615,E2 7647.615} C_VEL
LIN {X 0,Y 144.341,Z 1148.867,A -85,B 0,C 180,E1 7641.235,E2 7641.235} C_VEL
LIN {X 0,Y 145.482,Z 1147.292,A -85,B 0,C 180,E1 7634.044,E2 7634.044} C_VEL
LIN {X 0,Y 148.976,Z 1143.857,A -85,B 0,C 180,E1 7624.968,E2 7624.968} C_VEL
LIN {X 0,Y 154.492,Z 1139.262,A -85,B 0,C 180,E1 7617.069,E2 7617.069} C_VEL
LIN {X 0,Y 163.617,Z 1132.222,A -85,B 0,C 180,E1 7608.702,E2 7608.702} C_VEL
LIN {X 0,Y 173.863,Z 1124.425,A -85,B 0,C 180,E1 7602.111,E2 7602.111} C_VEL
LIN {X 0,Y 185.969,Z 1114.835,A -85,B 0,C 180,E1 7596.248,E2 7596.248} C_VEL
LIN {X 0,Y 198.992,Z 1104.07,A -85,B 0,C 180,E1 7591.331,E2 7591.331} C_VEL
LIN {X 0,Y 212.825,Z 1091.599,A -85,B 0,C 180,E1 7587.111,E2 7587.111} C_VEL
LIN {X 0,Y 226.9,Z 1077.944,A -85,B 0,C 180,E1 7583.57,E2 7583.57} C_VEL
LIN {X 0,Y 240.448,Z 1063.298,A -85,B 0,C 180,E1 7580.672,E2 7580.672} C_VEL
LIN {X 0,Y 254.567,Z 1046.506,A -85,B 0,C 180,E1 7578.077,E2 7578.077} C_VEL
LIN {X 0,Y 267.337,Z 1029.379,A -85,B 0,C 180,E1 7576.014,E2 7576.014} C_VEL
LIN {X 0,Y 280.444,Z 1009.442,A -85,B 0,C 180,E1 7574.128,E2 7574.128} C_VEL
LIN {X 0,Y 291.643,Z 989.988,A -85,B 0,C 180,E1 7572.675,E2 7572.675} C_VEL
LIN {X 0,Y 301.635,Z 969.551,A -85,B 0,C 180,E1 7571.472,E2 7571.472} C_VEL
LIN {X 0,Y 310.168,Z 949.328,A -85,B 0,C 180,E1 7570.518,E2 7570.518} C_VEL
LIN {X 0,Y 317.292,Z 928.576,A -85,B 0,C 180,E1 7569.745,E2 7569.745} C_VEL
LIN {X 0,Y 323.522,Z 906.327,A -85,B 0,C 180,E1 7569.095,E2 7569.095} C_VEL
LIN {X 0,Y 328.149,Z 883.764,A -85,B 0,C 180,E1 7568.606,E2 7568.606} C_VEL
LIN {X 0,Y 332.116,Z 854.293,A -85,B 0,C 180,E1 7568.093,E2 7568.093} C_VEL
LIN {X 0,Y 342.242,Z 763.461,A -85,B 0,C 180,E1 7566.572,E2 7566.572} C_VEL
LIN {X 0,Y 340.817,Z 758.941,A -85,B 0,C 180,E1 7561.682,E2 7561.682} C_VEL
LIN {X 0,Y 340.847,Z 759.124,A -85,B 0,C 180,E1 7558.488,E2 7558.488} C_VEL
LIN {X 0,Y 342.257,Z 763.506,A -85,B 0,C 180,E1 7553.879,E2 7553.879} C_VEL
LIN {X 0,Y 342.261,Z 764.015,A -85,B 0,C 180,E1 7553.78,E2 7553.78} C_VEL
LIN {X 0,Y 341.266,Z 772.878,A -85,B 0,C 180,E1 7553.632,E2 7553.632} C_VEL
LIN {X 0,Y 340.289,Z 780.579,A -85,B 0,C 180,E1 7553.669,E2 7553.669} C_VEL
LIN {X 0,Y 337.281,Z 801.187,A -85,B 0,C 180,E1 7554.388,E2 7554.388} C_VEL
LIN {X 0,Y 336.453,Z 807.796,A -85,B 0,C 180,E1 7554.409,E2 7554.409} C_VEL
LIN {X 0,Y 327.95,Z 880.365,A -85,B 0,C 180,E1 7553.221,E2 7553.221} C_VEL
LIN {X 0,Y 323.405,Z 903.824,A -85,B 0,C 180,E1 7552.786,E2 7552.786} C_VEL
LIN {X 0,Y 317.416,Z 926.656,A -85,B 0,C 180,E1 7552.288,E2 7552.288} C_VEL
LIN {X 0,Y 310.691,Z 946.613,A -85,B 0,C 180,E1 7551.725,E2 7551.725} C_VEL
LIN {X 0,Y 301.753,Z 968.786,A -85,B 0,C 180,E1 7550.902,E2 7550.902} C_VEL
LIN {X 0,Y 291.965,Z 989.029,A -85,B 0,C 180,E1 7549.922,E2 7549.922} C_VEL
LIN {X 0,Y 279.989,Z 1010.341,A -85,B 0,C 180,E1 7548.596,E2 7548.596} C_VEL
LIN {X 0,Y 268.195,Z 1028.638,A -85,B 0,C 180,E1 7547.135,E2 7547.135} C_VEL
LIN {X 0,Y 254.396,Z 1047.443,A -85,B 0,C 180,E1 7545.207,E2 7545.207} C_VEL
LIN {X 0,Y 240.515,Z 1064.416,A -85,B 0,C 180,E1 7542.968,E2 7542.968} C_VEL
LIN {X 0,Y 226.219,Z 1079.927,A -85,B 0,C 180,E1 7540.293,E2 7540.293} C_VEL
LIN {X 0,Y 211.72,Z 1094.409,A -85,B 0,C 180,E1 7537.057,E2 7537.057} C_VEL
LIN {X 0,Y 197.245,Z 1107.482,A -85,B 0,C 180,E1 7533.146,E2 7533.146} C_VEL
LIN {X 0,Y 182.471,Z 1119.956,A -85,B 0,C 180,E1 7528.138,E2 7528.138} C_VEL
LIN {X 0,Y 169.844,Z 1129.975,A -85,B 0,C 180,E1 7522.63,E2 7522.63} C_VEL
LIN {X 0,Y 157.438,Z 1139.537,A -85,B 0,C 180,E1 7515.339,E2 7515.339} C_VEL
LIN {X 0,Y 148.424,Z 1146.602,A -85,B 0,C 180,E1 7507.808,E2 7507.808} C_VEL
LIN {X 0,Y 141.401,Z 1152.524,A -85,B 0,C 180,E1 7498.739,E2 7498.739} C_VEL
LIN {X 0,Y 137.645,Z 1156.478,A -85,B 0,C 180,E1 7489.962,E2 7489.962} C_VEL
LIN {X 0,Y 136.154,Z 1158.949,A -85,B 0,C 180,E1 7481.006,E2 7481.006} C_VEL
LIN {X 0,Y 136.041,Z 1159.886,A -85,B 0,C 180,E1 7474.214,E2 7474.214} C_VEL
LIN {X 0,Y 136.071,Z 1160.032,A -85,B 0,C 180,E1 7468.315,E2 7468.315} C_VEL
LIN {X 0,Y 136.063,Z 1159.382,A -85,B 0,C 180,E1 7461.548,E2 7461.548} C_VEL
LIN {X 0,Y 136.685,Z 1157.783,A -85,B 0,C 180,E1 7454.296,E2 7454.296} C_VEL
LIN {X 0,Y 139.301,Z 1154.595,A -85,B 0,C 180,E1 7445.397,E2 7445.397} C_VEL
LIN {X 0,Y 144.688,Z 1149.6,A -85,B 0,C 180,E1 7436.437,E2 7436.437} C_VEL
LIN {X 0,Y 152.854,Z 1143.093,A -85,B 0,C 180,E1 7428.147,E2 7428.147} C_VEL
LIN {X 0,Y 163.602,Z 1134.724,A -85,B 0,C 180,E1 7420.725,E2 7420.725} C_VEL
LIN {X 0,Y 175.967,Z 1125.149,A -85,B 0,C 180,E1 7414.521,E2 7414.521} C_VEL
LIN {X 0,Y 190.027,Z 1113.574,A -85,B 0,C 180,E1 7409.138,E2 7409.138} C_VEL
LIN {X 0,Y 205.509,Z 1099.99,A -85,B 0,C 180,E1 7404.519,E2 7404.519} C_VEL
LIN {X 0,Y 219.844,Z 1086.322,A -85,B 0,C 180,E1 7401.056,E2 7401.056} C_VEL
LIN {X 0,Y 234.981,Z 1070.363,A -85,B 0,C 180,E1 7398.006,E2 7398.006} C_VEL
LIN {X 0,Y 249.143,Z 1053.95,A -85,B 0,C 180,E1 7395.596,E2 7395.596} C_VEL
LIN {X 0,Y 262.81,Z 1035.974,A -85,B 0,C 180,E1 7393.575,E2 7393.575} C_VEL
LIN {X 0,Y 275.881,Z 1016.701,A -85,B 0,C 180,E1 7391.886,E2 7391.886} C_VEL
LIN {X 0,Y 286.876,Z 998.138,A -85,B 0,C 180,E1 7390.618,E2 7390.618} C_VEL
LIN {X 0,Y 298.012,Z 976.452,A -85,B 0,C 180,E1 7389.456,E2 7389.456} C_VEL
LIN {X 0,Y 306.449,Z 957.16,A -85,B 0,C 180,E1 7388.652,E2 7388.652} C_VEL
LIN {X 0,Y 314.713,Z 934.45,A -85,B 0,C 180,E1 7387.921,E2 7387.921} C_VEL
LIN {X 0,Y 321.16,Z 912.442,A -85,B 0,C 180,E1 7387.393,E2 7387.393} C_VEL
LIN {X 0,Y 326.223,Z 889.013,A -85,B 0,C 180,E1 7386.939,E2 7386.939} C_VEL
LIN {X 0,Y 329.809,Z 864.628,A -85,B 0,C 180,E1 7386.519,E2 7386.519} C_VEL
LIN {X 0,Y 340.525,Z 770.121,A -85,B 0,C 180,E1 7384.977,E2 7384.977} C_VEL
LIN {X 0,Y 339.609,Z 766.796,A -85,B 0,C 180,E1 7381.18,E2 7381.18} C_VEL
LIN {X 0,Y 339.659,Z 767.018,A -85,B 0,C 180,E1 7377.806,E2 7377.806} C_VEL
LIN {X 0,Y 340.461,Z 770.244,A -85,B 0,C 180,E1 7374.541,E2 7374.541} C_VEL
LIN {X 0,Y 328.142,Z 876.273,A -85,B 0,C 180,E1 7372.823,E2 7372.823} C_VEL
LIN {X 0,Y 323.739,Z 899.541,A -85,B 0,C 180,E1 7372.373,E2 7372.373} C_VEL
LIN {X 0,Y 318.191,Z 921.331,A -85,B 0,C 180,E1 7371.827,E2 7371.827} C_VEL
LIN {X 0,Y 311.157,Z 942.566,A -85,B 0,C 180,E1 7371.127,E2 7371.127} C_VEL
LIN {X 0,Y 302.837,Z 963.566,A -85,B 0,C 180,E1 7370.248,E2 7370.248} C_VEL
LIN {X 0,Y 293.174,Z 983.702,A -85,B 0,C 180,E1 7369.181,E2 7369.181} C_VEL
LIN {X 0,Y 282.265,Z 1003.465,A -85,B 0,C 180,E1 7367.872,E2 7367.872} C_VEL
LIN {X 0,Y 270.608,Z 1021.664,A -85,B 0,C 180,E1 7366.352,E2 7366.352} C_VEL
LIN {X 0,Y 256.974,Z 1040.47,A -85,B 0,C 180,E1 7364.368,E2 7364.368} C_VEL
LIN {X 0,Y 244.089,Z 1056.201,A -85,B 0,C 180,E1 7362.251,E2 7362.251} C_VEL
LIN {X 0,Y 229.507,Z 1072.153,A -85,B 0,C 180,E1 7359.5,E2 7359.5} C_VEL
LIN {X 0,Y 215.891,Z 1085.621,A -85,B 0,C 180,E1 7356.494,E2 7356.494} C_VEL
LIN {X 0,Y 200.699,Z 1099.239,A -85,B 0,C 180,E1 7352.473,E2 7352.473} C_VEL
LIN {X 0,Y 186.598,Z 1110.925,A -85,B 0,C 180,E1 7347.848,E2 7347.848} C_VEL
LIN {X 0,Y 173.127,Z 1121.149,A -85,B 0,C 180,E1 7342.252,E2 7342.252} C_VEL
LIN {X 0,Y 161,Z 1130.014,A -85,B 0,C 180,E1 7335.578,E2 7335.578} C_VEL
LIN {X 0,Y 151.154,Z 1136.992,A -85,B 0,C 180,E1 7328.077,E2 7328.077} C_VEL
LIN {X 0,Y 143.114,Z 1142.916,A -85,B 0,C 180,E1 7318.821,E2 7318.821} C_VEL
LIN {X 0,Y 138.903,Z 1146.396,A -85,B 0,C 180,E1 7310.645,E2 7310.645} C_VEL
LIN {X 0,Y 136.642,Z 1148.84,A -85,B 0,C 180,E1 7301.322,E2 7301.322} C_VEL
LIN {X 0,Y 136.107,Z 1149.723,A -85,B 0,C 180,E1 7293.792,E2 7293.792} C_VEL
LIN {X 0,Y 136.091,Z 1149.793,A -85,B 0,C 180,E1 7287.474,E2 7287.474} C_VEL
LIN {X 0,Y 136.394,Z 1149.169,A -85,B 0,C 180,E1 7280.72,E2 7280.72} C_VEL
LIN {X 0,Y 137.8,Z 1147.489,A -85,B 0,C 180,E1 7272.694,E2 7272.694} C_VEL
LIN {X 0,Y 141.811,Z 1143.975,A -85,B 0,C 180,E1 7263.177,E2 7263.177} C_VEL
LIN {X 0,Y 148,Z 1139.326,A -85,B 0,C 180,E1 7254.954,E2 7254.954} C_VEL
LIN {X 0,Y 157.498,Z 1132.531,A -85,B 0,C 180,E1 7246.716,E2 7246.716} C_VEL
LIN {X 0,Y 168.424,Z 1124.734,A -85,B 0,C 180,E1 7240.021,E2 7240.021} C_VEL
LIN {X 0,Y 181.195,Z 1115.144,A -85,B 0,C 180,E1 7234.135,E2 7234.135} C_VEL
LIN {X 0,Y 195.314,Z 1103.988,A -85,B 0,C 180,E1 7229.1,E2 7229.1} C_VEL
LIN {X 0,Y 209.601,Z 1091.541,A -85,B 0,C 180,E1 7224.994,E2 7224.994} C_VEL
LIN {X 0,Y 224.54,Z 1077.418,A -85,B 0,C 180,E1 7221.462,E2 7221.462} C_VEL
LIN {X 0,Y 238.513,Z 1062.69,A -85,B 0,C 180,E1 7218.666,E2 7218.666} C_VEL
LIN {X 0,Y 253.846,Z 1044.655,A -85,B 0,C 180,E1 7216.039,E2 7216.039} C_VEL
LIN {X 0,Y 266.977,Z 1027.273,A -85,B 0,C 180,E1 7214.075,E2 7214.075} C_VEL
LIN {X 0,Y 279.476,Z 1008.285,A -85,B 0,C 180,E1 7212.395,E2 7212.395} C_VEL
LIN {X 0,Y 290.819,Z 988.706,A -85,B 0,C 180,E1 7211.017,E2 7211.017} C_VEL
LIN {X 0,Y 300.727,Z 968.568,A -85,B 0,C 180,E1 7209.899,E2 7209.899} C_VEL
LIN {X 0,Y 309.727,Z 947.075,A -85,B 0,C 180,E1 7208.949,E2 7208.949} C_VEL
LIN {X 0,Y 316.494,Z 927.418,A -85,B 0,C 180,E1 7208.266,E2 7208.266} C_VEL
LIN {X 0,Y 322.88,Z 904.283,A -85,B 0,C 180,E1 7207.637,E2 7207.637} C_VEL
LIN {X 0,Y 327.287,Z 882.723,A -85,B 0,C 180,E1 7207.196,E2 7207.196} C_VEL
LIN {X 0,Y 331.418,Z 851.611,A -85,B 0,C 180,E1 7206.674,E2 7206.674} C_VEL
LIN {X 0,Y 340.675,Z 770.233,A -85,B 0,C 180,E1 7205.347,E2 7205.347} C_VEL
LIN {X 0,Y 339.82,Z 766.87,A -85,B 0,C 180,E1 7201.518,E2 7201.518} C_VEL
LIN {X 0,Y 339.849,Z 767.012,A -85,B 0,C 180,E1 7198.652,E2 7198.652} C_VEL
LIN {X 0,Y 340.715,Z 770.435,A -85,B 0,C 180,E1 7195.015,E2 7195.015} C_VEL
LIN {X 0,Y 336.453,Z 807.796,A -85,B 0,C 180,E1 7194.409,E2 7194.409} C_VEL
LIN {X 0,Y 335.476,Z 815.496,A -85,B 0,C 180,E1 7194.454,E2 7194.454} C_VEL
LIN {X 0,Y 332.525,Z 836.092,A -85,B 0,C 180,E1 7195.195,E2 7195.195} C_VEL
LIN {X 0,Y 331.698,Z 842.7,A -85,B 0,C 180,E1 7195.221,E2 7195.221} C_VEL
LIN {X 0,Y 326.726,Z 882.379,A -85,B 0,C 180,E1 7194.582,E2 7194.582} C_VEL
LIN {X 0,Y 322.101,Z 905.245,A -85,B 0,C 180,E1 7194.172,E2 7194.172} C_VEL
LIN {X 0,Y 315.339,Z 929.747,A -85,B 0,C 180,E1 7193.651,E2 7193.651} C_VEL
LIN {X 0,Y 308.563,Z 949.205,A -85,B 0,C 180,E1 7193.114,E2 7193.114} C_VEL
LIN {X 0,Y 299.154,Z 971.518,A -85,B 0,C 180,E1 7192.302,E2 7192.302} C_VEL
LIN {X 0,Y 288.995,Z 991.923,A -85,B 0,C 180,E1 7191.337,E2 7191.337} C_VEL
LIN {X 0,Y 277.093,Z 1012.261,A -85,B 0,C 180,E1 7190.092,E2 7190.092} C_VEL
LIN {X 0,Y 264.658,Z 1031,A -85,B 0,C 180,E1 7188.629,E2 7188.629} C_VEL
LIN {X 0,Y 251.07,Z 1048.821,A -85,B 0,C 180,E1 7186.828,E2 7186.828} C_VEL
LIN {X 0,Y 236.073,Z 1066.432,A -85,B 0,C 180,E1 7184.525,E2 7184.525} C_VEL
LIN {X 0,Y 221.859,Z 1081.334,A -85,B 0,C 180,E1 7181.974,E2 7181.974} C_VEL
LIN {X 0,Y 205.375,Z 1096.95,A -85,B 0,C 180,E1 7178.415,E2 7178.415} C_VEL
LIN {X 0,Y 190.574,Z 1109.761,A -85,B 0,C 180,E1 7174.476,E2 7174.476} C_VEL
LIN {X 0,Y 176.01,Z 1121.288,A -85,B 0,C 180,E1 7169.631,E2 7169.631} C_VEL
LIN {X 0,Y 162.418,Z 1131.544,A -85,B 0,C 180,E1 7163.749,E2 7163.749} C_VEL
LIN {X 0,Y 150.123,Z 1140.32,A -85,B 0,C 180,E1 7156.549,E2 7156.549} C_VEL
LIN {X 0,Y 139.959,Z 1147.734,A -85,B 0,C 180,E1 7147.906,E2 7147.906} C_VEL
LIN {X 0,Y 133.416,Z 1152.865,A -85,B 0,C 180,E1 7139.151,E2 7139.151} C_VEL
LIN {X 0,Y 129.32,Z 1156.885,A -85,B 0,C 180,E1 7128.948,E2 7128.948} C_VEL
LIN {X 0,Y 128.12,Z 1158.868,A -85,B 0,C 180,E1 7120.339,E2 7120.339} C_VEL
LIN {X 0,Y 128.047,Z 1159.637,A -85,B 0,C 180,E1 7113.581,E2 7113.581} C_VEL
LIN {X 0,Y 128.065,Z 1159.708,A -85,B 0,C 180,E1 7107.762,E2 7107.762} C_VEL
LIN {X 0,Y 128.082,Z 1159.079,A -85,B 0,C 180,E1 7101.017,E2 7101.017} C_VEL
LIN {X 0,Y 128.921,Z 1157.354,A -85,B 0,C 180,E1 7092.859,E2 7092.859} C_VEL
LIN {X 0,Y 132.256,Z 1153.916,A -85,B 0,C 180,E1 7083.024,E2 7083.024} C_VEL
LIN {X 0,Y 138.512,Z 1148.756,A -85,B 0,C 180,E1 7073.705,E2 7073.705} C_VEL
LIN {X 0,Y 148.146,Z 1141.72,A -85,B 0,C 180,E1 7064.873,E2 7064.873} C_VEL
LIN {X 0,Y 159.422,Z 1133.574,A -85,B 0,C 180,E1 7057.79,E2 7057.79} C_VEL
LIN {X 0,Y 174.031,Z 1122.722,A -85,B 0,C 180,E1 7051.122,E2 7051.122} C_VEL
LIN {X 0,Y 188.632,Z 1111.255,A -85,B 0,C 180,E1 7046.1,E2 7046.1} C_VEL
LIN {X 0,Y 203.772,Z 1098.247,A -85,B 0,C 180,E1 7041.968,E2 7041.968} C_VEL
LIN {X 0,Y 218.587,Z 1084.501,A -85,B 0,C 180,E1 7038.674,E2 7038.674} C_VEL
LIN {X 0,Y 233.848,Z 1068.64,A -85,B 0,C 180,E1 7035.837,E2 7035.837} C_VEL
LIN {X 0,Y 248.911,Z 1051.299,A -85,B 0,C 180,E1 7033.472,E2 7033.472} C_VEL
LIN {X 0,Y 261.957,Z 1034.37,A -85,B 0,C 180,E1 7031.696,E2 7031.696} C_VEL
LIN {X 0,Y 275.744,Z 1014.092,A -85,B 0,C 180,E1 7030.047,E2 7030.047} C_VEL
LIN {X 0,Y 287.36,Z 994.558,A -85,B 0,C 180,E1 7028.817,E2 7028.817} C_VEL
LIN {X 0,Y 297.731,Z 974.119,A -85,B 0,C 180,E1 7027.819,E2 7027.819} C_VEL
LIN {X 0,Y 306.951,Z 952.985,A -85,B 0,C 180,E1 7027.016,E2 7027.016} C_VEL
LIN {X 0,Y 314.472,Z 931.763,A -85,B 0,C 180,E1 7026.404,E2 7026.404} C_VEL
LIN {X 0,Y 321.021,Z 909.006,A -85,B 0,C 180,E1 7025.904,E2 7025.904} C_VEL
LIN {X 0,Y 325.796,Z 886.252,A -85,B 0,C 180,E1 7025.489,E2 7025.489} C_VEL
LIN {X 0,Y 330.032,Z 855.236,A -85,B 0,C 180,E1 7024.981,E2 7024.981} C_VEL
LIN {X 0,Y 339.063,Z 777.082,A -85,B 0,C 180,E1 7023.719,E2 7023.719} C_VEL
LIN {X 0,Y 338.611,Z 774.727,A -85,B 0,C 180,E1 7021.015,E2 7021.015} C_VEL
LIN {X 0,Y 338.659,Z 774.908,A -85,B 0,C 180,E1 7017.969,E2 7017.969} C_VEL
LIN {X 0,Y 339.021,Z 777.18,A -85,B 0,C 180,E1 7015.782,E2 7015.782} C_VEL
LIN {X 0,Y 327.239,Z 876.594,A -85,B 0,C 180,E1 7014.213,E2 7014.213} C_VEL
LIN {X 0,Y 322.774,Z 899.855,A -85,B 0,C 180,E1 7013.782,E2 7013.782} C_VEL
LIN {X 0,Y 317.151,Z 921.643,A -85,B 0,C 180,E1 7013.261,E2 7013.261} C_VEL
LIN {X 0,Y 309.934,Z 943.107,A -85,B 0,C 180,E1 7012.585,E2 7012.585} C_VEL
LIN {X 0,Y 301.108,Z 964.878,A -85,B 0,C 180,E1 7011.71,E2 7011.71} C_VEL
LIN {X 0,Y 291.303,Z 984.903,A -85,B 0,C 180,E1 7010.688,E2 7010.688} C_VEL
LIN {X 0,Y 279.755,Z 1005.23,A -85,B 0,C 180,E1 7009.382,E2 7009.382} C_VEL
LIN {X 0,Y 268.128,Z 1022.966,A -85,B 0,C 180,E1 7007.946,E2 7007.946} C_VEL
LIN {X 0,Y 254.01,Z 1041.876,A -85,B 0,C 180,E1 7006.004,E2 7006.004} C_VEL
LIN {X 0,Y 240.949,Z 1057.403,A -85,B 0,C 180,E1 7003.969,E2 7003.969} C_VEL
LIN {X 0,Y 225.923,Z 1073.296,A -85,B 0,C 180,E1 7001.281,E2 7001.281} C_VEL
LIN {X 0,Y 211.133,Z 1087.447,A -85,B 0,C 180,E1 6998.158,E2 6998.158} C_VEL
LIN {X 0,Y 195.892,Z 1100.474,A -85,B 0,C 180,E1 6994.287,E2 6994.287} C_VEL
LIN {X 0,Y 180.925,Z 1112.272,A -85,B 0,C 180,E1 6989.557,E2 6989.557} C_VEL
LIN {X 0,Y 167.614,Z 1121.867,A -85,B 0,C 180,E1 6984.222,E2 6984.222} C_VEL
LIN {X 0,Y 154.25,Z 1131.009,A -85,B 0,C 180,E1 6977.096,E2 6977.096} C_VEL
LIN {X 0,Y 144.222,Z 1137.662,A -85,B 0,C 180,E1 6969.631,E2 6969.631} C_VEL
LIN {X 0,Y 135.687,Z 1143.422,A -85,B 0,C 180,E1 6960.073,E2 6960.073} C_VEL
LIN {X 0,Y 130.966,Z 1147.003,A -85,B 0,C 180,E1 6951.029,E2 6951.029} C_VEL
LIN {X 0,Y 128.627,Z 1149.257,A -85,B 0,C 180,E1 6941.207,E2 6941.207} C_VEL
LIN {X 0,Y 128.107,Z 1150.044,A -85,B 0,C 180,E1 6933.581,E2 6933.581} C_VEL
LIN {X 0,Y 128.097,Z 1150.094,A -85,B 0,C 180,E1 6927.317,E2 6927.317} C_VEL
LIN {X 0,Y 128.46,Z 1149.47,A -85,B 0,C 180,E1 6920.141,E2 6920.141} C_VEL
LIN {X 0,Y 130.058,Z 1147.794,A -85,B 0,C 180,E1 6911.628,E2 6911.628} C_VEL
LIN {X 0,Y 134.541,Z 1144.282,A -85,B 0,C 180,E1 6901.601,E2 6901.601} C_VEL
LIN {X 0,Y 141.329,Z 1139.634,A -85,B 0,C 180,E1 6893.034,E2 6893.034} C_VEL
LIN {X 0,Y 151.58,Z 1132.841,A -85,B 0,C 180,E1 6884.571,E2 6884.571} C_VEL
LIN {X 0,Y 163.3,Z 1124.992,A -85,B 0,C 180,E1 6877.756,E2 6877.756} C_VEL
LIN {X 0,Y 176.683,Z 1115.453,A -85,B 0,C 180,E1 6871.913,E2 6871.913} C_VEL
LIN {X 0,Y 190.922,Z 1104.686,A -85,B 0,C 180,E1 6867.091,E2 6867.091} C_VEL
LIN {X 0,Y 205.462,Z 1092.536,A -85,B 0,C 180,E1 6863.112,E2 6863.112} C_VEL
LIN {X 0,Y 220.837,Z 1078.556,A -85,B 0,C 180,E1 6859.655,E2 6859.655} C_VEL
LIN {X 0,Y 235.16,Z 1063.907,A -85,B 0,C 180,E1 6856.931,E2 6856.931} C_VEL
LIN {X 0,Y 249.949,Z 1047.151,A -85,B 0,C 180,E1 6854.521,E2 6854.521} C_VEL
LIN {X 0,Y 263.043,Z 1030.341,A -85,B 0,C 180,E1 6852.643,E2 6852.643} C_VEL
LIN {X 0,Y 276.475,Z 1010.769,A -85,B 0,C 180,E1 6850.928,E2 6850.928} C_VEL
LIN {X 0,Y 287.528,Z 992.316,A -85,B 0,C 180,E1 6849.65,E2 6849.65} C_VEL
LIN {X 0,Y 298.237,Z 971.443,A -85,B 0,C 180,E1 6848.505,E2 6848.505} C_VEL
